# B&R Automation Studio project NAEUL004C00R13L518F00 (part 72)

#### Act_InitLocal.st
```iecst
(** 2019-04-16 **)
ACTION Act_InitLocal:

	//Input Reference Link To Local Variable
	p_udiRstErr ACCESS ADR(udiRstErr);
	p_bEn ACCESS ADR(bEn);
	p_bDis ACCESS ADR(bDis);
	p_bRun ACCESS ADR(bRun);
	p_bStop ACCESS ADR(bStop);
	p_bStep ACCESS ADR(bStep);

	p_sProgNm ACCESS ADR(sProgNm);
	p_bNtSettingsLoadDone ACCESS ADR(bNtSettingsLoadDone);

	p_usiMagConv ACCESS ADR(usiMagConv);
	p_bInfoEn ACCESS ADR(bInfoEn);

	pa_bMagDis ACCESS ADR(a_bMagDis);
	pa_bMagRej ACCESS ADR(a_bMagRej);
	p_bUSAllow ACCESS ADR(bUSAllow);

	p_bAllwChgWidth  ACCESS ADR(bAllwChgWidth);
	p_bAllwChgSlot ACCESS ADR(bAllwChgSlot);

	p_bNewMag ACCESS ADR(bNewMag);
	p_bRlsMag ACCESS ADR(bRlsMag);

	p_bConvInitDone ACCESS ADR(bConvInitDone);
	p_bConvHvBrd ACCESS ADR(bConvHvBrd);
	p_bConvGdBrd ACCESS ADR(bConvGdBrd);

	p_tyBufferStat1 ACCESS ADR(tyBufferStat1);
	p_tyBufferStat2 ACCESS ADR(tyBufferStat2);
	p_tyBufferStat3 ACCESS ADR(tyBufferStat3);

	p_bMagClampRS1 ACCESS ADR(bMagClampRS1);
	p_bMagClampRS2 ACCESS ADR(bMagClampRS2);
	p_bMagClampRS3 ACCESS ADR(bMagClampRS3);

	p_bMagEntrySen1 ACCESS ADR(bMagEntrySen1);
	p_bMagEntrySen2 ACCESS ADR(bMagEntrySen2);
	p_bMagEntrySen3 ACCESS ADR(bMagEntrySen3);

	p_bMagPresentSen1 ACCESS ADR(bMagPresentSen1);
	p_bMagPresentSen2 ACCESS ADR(bMagPresentSen2);
	p_bMagPresentSen3 ACCESS ADR(bMagPresentSen3);

	p_bBufferMagPresent1 ACCESS ADR(bBufferMagPresent1);
	p_bBufferMagPresent2 ACCESS ADR(bBufferMagPresent2);
	p_bBufferMagPresent3 ACCESS ADR(bBufferMagPresent3);

	p_dtBufferMagPresentTm1 ACCESS ADR(dtBufferMagPresentTm1);
	p_dtBufferMagPresentTm2 ACCESS ADR(dtBufferMagPresentTm2);
	p_dtBufferMagPresentTm3 ACCESS ADR(dtBufferMagPresentTm3);

	p_eBufferStat ACCESS ADR(eBufferStat);
	p_eBufferStatus ACCESS ADR(eBufferStatus);

	p_eMagConv2ClpStat ACCESS ADR(eMagConv2ClpStat);
	p_eMagConv2ClpStatus ACCESS ADR(eMagConv2ClpStatus);
	p_bMagConv2ClpHvMag ACCESS ADR(bMagConv2ClpHvMag);

	p_eUSSMEMAStat ACCESS ADR(eUSSMEMAStat);
	p_eUSSMEMAStatus ACCESS ADR(eUSSMEMAStatus);
	p_bUSSMEMATransporting ACCESS ADR(bUSSMEMATransporting);
	p_bUSSMEMAConvStart ACCESS ADR(bUSSMEMAConvStart);
	p_bUSSMEMAConvStop ACCESS ADR(bUSSMEMAConvStop);

	p_eAGVMagStat ACCESS ADR(eAGVMagStat);
	p_eAGVMagStatus ACCESS ADR(eAGVMagStatus);
	p_bAGVMagMcRunRdy ACCESS ADR(bAGVMagMcRunRdy);
	p_tyAGVToDTMag ACCESS ADR(tyAGVToDualMag);

	p_dtOpsMagConvUL3AcptTm ACCESS ADR(dtMagConvAcptTm);
	p_iOpsMagConvUL3MESAcptCond ACCESS ADR(iMagMESAcptCond);
END_ACTION
```

#### Act_Link.st
```iecst
(** 2018-12-11 **)
ACTION Act_Link:

	//Clamp RS
	p_bMagClampRS1 		:= (p_bLinkFixedMagClampRS1 AND p_bLinkRmtMagClampRS1) OR p_bLinkNewMagVerified1;
	p_bMagClampRS2		:= (p_bLinkFixedMagClampRS2 AND p_bLinkRmtMagClampRS2) OR p_bLinkNewMagVerified2;
	p_bMagClampRS3		:= (p_bLinkFixedMagClampRS3 AND p_bLinkRmtMagClampRS3) OR bNewMagVerified;

	//Mag Exchange Mode
	CASE p_eLinkMcParamMagExMode OF
		McSetMagXcAutoManMode:
			bMagManEx := TRUE;
			bMagAutoEx := TRUE;

		McSetMagXcAutoMode:
			bMagManEx := FALSE;
			bMagAutoEx := TRUE;

		McSetMagXcManMode:
			bMagManEx := TRUE;
			bMagAutoEx := FALSE;

	END_CASE

	//New magazine auto detection at inlet sensor
	fbMagAutoDetTm(IN := p_bLinkDIMagEntrySen OR p_bLinkDIMagPresentSen3, PT := DINT_TO_TIME(p_bLinkMcParamMagAutoDetTm));
	IF fbMagAutoDetTm.Q AND bMagManEx THEN
		bNewMagAutoDetected := TRUE;
	ELSE
		bNewMagAutoDetected := FALSE;
	END_IF

	IF p_bLinkNtParamMagModelAutoVerify THEN
		IF p_bLinkMagRcpCurrRcpMagModel = 0  //CAB706.2
			AND p_bDIMagConvHeightSen = TRUE
			AND p_bDIMagConvSelUnclampRS = FALSE
			AND p_bDIMagConvCAB717Sen = FALSE
			AND p_bDIMagConvSmallSen
			AND ((NOT p_bMagAWCloseLimit AND NOT  p_bMagAWOpenLimit) OR p_tyBufferStat3.bBffrMty = FALSE)
			THEN
			bNewMagVerified:= TRUE;

		ELSIF  p_bLinkMagRcpCurrRcpMagModel = 1 //CAB716.2
			AND p_bDIMagConvHeightSen = FALSE
			AND p_bDIMagConvSelUnclampRS = FALSE
			AND p_bDIMagConvCAB717Sen = FALSE
			AND p_bDIMagConvSmallSen
			AND ((NOT p_bMagAWCloseLimit AND NOT  p_bMagAWOpenLimit) OR p_tyBufferStat3.bBffrMty = FALSE)
			THEN
			bNewMagVerified:= TRUE;

		ELSIF  p_bLinkMagRcpCurrRcpMagModel = 2 //CAB717.2
			AND p_bDIMagConvHeightSen = FALSE
			AND p_bDIMagConvSelUnclampRS
			AND p_bDIMagConvCAB717Sen
			AND p_bDIMagConvLargeSen
			AND ((NOT p_bMagAWCloseLimit AND NOT  p_bMagAWOpenLimit) OR p_tyBufferStat3.bBffrMty = FALSE)
			THEN
			bNewMagVerified:= TRUE;
		ELSE
			bNewMagVerified:= FALSE;
		END_IF
	ELSE
		bNewMagVerified:= TRUE;
	END_IF

	bAIVInPos := p_tyAGVToDTMag.bVEHInPos3 OR p_bDISOTRcv;

	IF p_bBufferMagRemoved THEN
		bManualUnloadMag := FALSE;
	END_IF

	IF bAutoRcpEn THEN
		p_bUSAllow :=  ( NOT(p_bNtParamAutoRcpF1ArbitraryType) AND NOT(p_bMagPropDiffBlk) ) AND
						(p_bNtParamAutoRcpF1ArbitraryType AND p_sProdRcpCurrRcp1Name = p_sProdRcpCurrRcp2Name)	;
		p_bAllwChgWidth := p_bChgMagWidth AND NOT(p_bNtParamAutoRcpF1ArbitraryType);
		p_bAllwChgSlot	:= p_bChgMagSlot AND NOT(p_bNtParamAutoRcpF1ArbitraryType);

	ELSE
		p_bUSAllow := p_sProdRcpCurrRcp1Name = p_sProdRcpCurrRcp2Name;
	END_IF

END_ACTION
```

#### Cyclic.st
```iecst
(** 2019-03-22 **)
PROGRAM _CYCLIC

	IF bInitDone = FALSE THEN
		bInitDone	:= TRUE;

		Act_InitLocal;
		Act_InitGlobal;

	ELSIF bInitialDone = FALSE THEN
		IF p_bNtSettingsLoadDone = TRUE THEN
			bInitialDone	:= TRUE;

			Act_Initial;
		END_IF

	ELSE

		Act_RstErr;
		Act_LinkEn;
		Act_Link;
		Act_Background;
		Act_Alarm;
		Act_AlarmInfo1;

	END_IF

END_PROGRAM
```

#### Init.st
```iecst
(** 2019-03-25 **)
PROGRAM _INIT

	(* Always Change If Project Change *)

	//Physical Configuration
	usiMagConv	:= 3;

	//Pass Address To Global Address For External Use
	//Action, State & Status

	//Alarm
	p_OpsMagConvUL3AlmData	:= ADR(tyAlmData);
	p_OpsMagConvUL3AlmData1	:= ADR(tyAlmData1);

	//Output
	p_OpsMagConvUL3StepTxt			:= ADR(sStepTxt);
	p_OpsMagConvUL3Paused			:= ADR(bPaused);

	p_OpsMagConvUL3BufferAct		:= ADR(eBufferAct);
	p_OpsMagConvUL3MagConv2ClpAct	:= ADR(eMagConv2ClpAct);
	p_OpsMagConvUL3USSMEMAAct		:= ADR(eUSSMEMAAct);
	p_OpsMagConvUL3AGVMagAct		:= ADR(eAGVMagAct);

	p_OpsMagConvUL3InitDone				:= ADR(bOpsInitDone);
	p_OpsMagConvUL3MagBffrAvl			:= ADR(bMagBffrAvl);
	p_OpsMagConvUL3NewMagAllw			:= ADR(bNewMagAllw);
	p_OpsMagConvUL3RlsMagAllw			:= ADR(bRlsMagAllw);
	p_OpsMagConvUL3EjectMESStep			:= ADR(bEjectMESStep); //MES
	p_OpsMagConvUL3EjectMagNotAllw		:= ADR(bEjectMagNotAllw); //MES
	p_OpsMagConvUL3StepMagExitedWait	:= ADR(bStepMagExitedWait);
	p_OpsMagConvUL3StepUSCom			:= ADR(bStepMagUSCom);
	p_OpsMagConvUL3StepPLCGrab			:= ADR(bStepPLCGrab);

	p_OpsMagConvUL3StepSelClampCtrl		:= ADR(eSelClampCtrl);
	p_OpsMagConvUL3NewMagVerified		:= ADR(bNewMagVerified);
	p_OpsMagConvUL3MagFullExit			:= ADR(bStepMagFullExit);
	p_OpsMagConvUL3IncorrectMagModel    := ADR(bIncorrectMagazineModel);
	p_OpsMagConvUL3MagSizeL    			:= ADR(bMagSizeLarge);

	p_OpsMagConvUL3SafetyBarAct			:= ADR(eSafetyBarAct);
	p_OpsMagConvUL3MagAWEngageAct		:= ADR(eMagAWEngageAct);
	p_OpsMagConvUL3MagAWAct				:= ADR(eMagAWAct);

	p_OpsMagConvUL3USSOTAct				:= ADR(eUSSOTAct);
	p_OpsMagConvUL3DSSOTAct				:= ADR(eDSSOTAct);

	p_OpsAGVCommRdy3					:= ADR(bAGVComm3Rdy);

	p_OpsMagConvUL3UnclmpDone			:= ADR(bPneuUnclmpDone);
	p_OpsMagConvUL3MagAllwGo			:= ADR(udiMagAllwGo);

	p_OpsMagConvUL3ReadRFID				:= ADR(bReadRFID);
	p_OpsMagConvUL3WriteRFID			:= ADR(bWriteRFID);
	p_OpsMagConvUL3AWDone			 	:= ADR(bStepOpsMagAWDone);
	p_OpsMagConvUL3SlotUpdtDone			:= ADR(bStepOpsPitchUpdated);
	(* Always Change If Project Change *)

	p_OpsMagConvUL3AcptTm				:= ADR(dtMagConvAcptTm);
	p_OpsMagConvUL3MESAcptCond 			:= ADR(iMagMESAcptCond);
	p_OpsMagConvUL3MagExitedWait 		:= ADR(bMagExitedWait);
END_PROGRAM
```

#### Act_OpsInitial.st - Do Not Change!!!
```iecst
(** 2019-01-16 **)
ACTION Act_OpsInitial:

	eOpsStep			:= MagConvULStepNA;
	eGotoOpsStep		:= MagConvULStepInitMag;

	bOpsInitDone		:= FALSE;
	bMagBffrAvl			:= FALSE;
	bNewMagAllw			:= FALSE;
	bRlsMagAllw			:= FALSE;
	bStepMagExitedWait	:= FALSE;
	bAGVComm3Rdy		:= FALSE;

END_ACTION
```

#### Act_OpsRun.st
```iecst
(** 2019-04-16 **)
ACTION Act_OpsRun:
	IF p_bOpsTravLifErrCmdUnclmp THEN //from travLif width chk error
		eMagConv2ClpAct :=	MagConv2ClpActStopClpr;

		IF (p_eMagConv2ClpStatus = Done AND p_eMagConv2ClpStat = MagConv2ClpActStopClpr) THEN

			eMagConv2ClpAct	:= MagConv2ClpActIdle;
			bPneuUnclmpDone := TRUE; //To TravLifUL
		END_IF
	END_IF

	Act_LogStep;

	IF eGotoOpsStep <> eOpsStep THEN

		fbWrongMagTm(IN:= FALSE);
		fbReadRFIDTO(IN:= FALSE);
		fbWriteRFIDTO(IN:= FALSE);
		CASE eGotoOpsStep OF
			MagConvULStepBffrStatChk:  //For Siemen, Enter Condition
				IF ((p_eCustomerReq = Siemens OR p_eCustomerReq = We_Fabricate) AND p_bMcParamMESEn) AND eOpsStep = MagConvULStepVerifyMag THEN
					IF ePrevStepBeforeMESStdBy = MagConvULStepMagExitMnl OR ePrevStepBeforeMESStdBy = MagConvULStepMagExitClampCtrl THEN
						eGotoOpsStep		:= MagConvULStepMagExtMESStdByChk;
						eOpsStep			:= MagConvULStepMagExtMESStdByChk;
					ELSIF  iMagMESAcptCond > 0 THEN
						eGotoOpsStep		:= MagConvULStepBffrStatChk;
						eOpsStep			:= MagConvULStepBffrStatChk;
					ELSIF iMagMESAcptCond < 0 THEN
						eGotoOpsStep		:= MagConvULStepMagExitClampCtrl;
						eOpsStep			:= MagConvULStepMagExitClampCtrl;
					ELSIF iMagMESAcptCond = 0 THEN
						eGotoOpsStep		:= MagConvULStepMagEntMESStdByChk;
						eOpsStep			:= MagConvULStepMagEntMESStdByChk;
					END_IF
				ELSE
					eOpsStep	:= eGotoOpsStep;
				END_IF
			MagConvULStepMagExitClampCtrl: //For Siemen, Bffr Full,Changover Mag, AGV Rdy,Reject Mag
				IF (p_eCustomerReq = Siemens AND p_bMcParamMESEn) AND (eOpsStep <> MagConvULStepMagExtMESStdByChk )
					AND (p_tyLocalBufferStat.bBffrFull OR pa_bMagChangeOverBlk[p_usiMagConv] = TRUE OR p_bDISOTAGVReady)
					AND NOT(iMagMESAcptCond < 0)THEN
					eOpsStep := MagConvULStepMagExtMESStdByChk;
					eGotoOpsStep := MagConvULStepMagExtMESStdByChk;
					ePrevStepBeforeMESStdBy := MagConvULStepMagExitClampCtrl;
				ELSE
					eOpsStep	:= eGotoOpsStep;
					ePrevStepBeforeMESStdBy	:= MagConvULStepNA;
				END_IF
			MagConvULStepMagExitMnl: //For Siemens, Manual Rls
				IF (p_eCustomerReq = Siemens AND p_bMcParamMESEn)
					AND (eOpsStep <> MagConvULStepMagExtMESStdByChk AND eOpsStep <> MagConvULStepMagFullDSComm
					AND eOpsStep <> MagConvULStepMagEntMESStdByChk AND eOpsStep <> MagConvULStepVerifyMag)
					THEN
					eOpsStep := MagConvULStepMagExtMESStdByChk;
					eGotoOpsStep := MagConvULStepMagExtMESStdByChk;
					ePrevStepBeforeMESStdBy := MagConvULStepMagExitMnl;
				ELSE
//					sStepTxt	:= 'Waiting for Shutter Close';
//					IF (p_bNtParamProjOutletShut3Prep AND p_bDIOutShutterClosedRS3) OR (NOT(p_bNtParamProjOutletShut3Prep) AND p_bDIOutShutterClosedRS) THEN
						eOpsStep	:= eGotoOpsStep;
						ePrevStepBeforeMESStdBy	:= MagConvULStepNA;
//					END_IF
				END_IF
			MagConvULStepSelClampCtrl:
				IF p_bMagOrientChkSenPrep THEN
					IF p_bMagHeightDetEn AND p_bMagHeightDetPrep THEN

						IF p_bMag3OrientationChkSen1 AND p_bMagHeightDetSen3 THEN // Magazine Type Check with height Detection Sensor
							eOpsStep := eGotoOpsStep;
						ELSE
							eMagConv2ClpAct :=	MagConv2ClpActStopClpr; //Unclamp First

							IF (p_eMagConv2ClpStatus = Done AND p_eMagConv2ClpStat = MagConv2ClpActStopClpr) THEN

								eMagConv2ClpAct	:= MagConv2ClpActIdle;

								eStatus		:= Error;
								udiStatus	:= 10011;	//Wrong Magazine Orientation Placed.
							END_IF
						END_IF

					ELSE

						IF p_bMag3OrientationChkSen1 AND NOT p_bMagHeightDetSen3 THEN //Without Check Height Detection Sensor
							eOpsStep := eGotoOpsStep;
						ELSE
							eMagConv2ClpAct :=	MagConv2ClpActStopClpr; //Unclamp First

							IF (p_eMagConv2ClpStatus = Done AND p_eMagConv2ClpStat = MagConv2ClpActStopClpr) THEN

								eMagConv2ClpAct	:= MagConv2ClpActIdle;

								eStatus		:= Error;
								udiStatus	:= 10011;	//Wrong Magazine Orientation Placed.
							END_IF
						END_IF

					END_IF
				ELSE
					eOpsStep	:= eGotoOpsStep;
				END_IF
			ELSE
				eOpsStep	:= eGotoOpsStep;

		END_CASE

	END_IF

	IF eOpsStep = eGotoOpsStep THEN

		IF bPaused = FALSE THEN

			CASE eOpsStep OF

				MagConvULStepInitMag:
					sStepTxt	:= 'Initializing Magazine';
					p_usiMagConv := 3;
					CASE p_usiMagConv OF
						1:
							p_tyLocalBufferStat ACCESS ADR(p_tyBufferStat1);
							p_bLocalMagEntrySen ACCESS ADR(p_bMagEntrySen1);
							p_bLocalBufferMagPresent ACCESS ADR(p_bBufferMagPresent1);
							p_dtLocalBufferMagPresentTm ACCESS ADR(p_dtBufferMagPresentTm1);
						2:
							p_tyLocalBufferStat ACCESS ADR(p_tyBufferStat2);
							p_bLocalMagEntrySen ACCESS ADR(p_bMagEntrySen2);
							p_bLocalBufferMagPresent ACCESS ADR(p_bBufferMagPresent2);
							p_dtLocalBufferMagPresentTm ACCESS ADR(p_dtBufferMagPresentTm2);
						3:
							p_tyLocalBufferStat ACCESS ADR(p_tyBufferStat3);
							p_bLocalMagEntrySen ACCESS ADR(p_bMagEntrySen3);
							p_bLocalBufferMagPresent ACCESS ADR(p_bBufferMagPresent3);
							p_dtLocalBufferMagPresentTm ACCESS ADR(p_dtBufferMagPresentTm3);
					END_CASE

//					IF bMagExitedWait THEN
//						eGotoOpsStep	:= MagConvULStepMagExitedWait;
//					ELSE
//						eGotoOpsStep	:= MagConvULStepInitMagConv;
//					END_IF

					IF p_bProjLifTravMnlLoad = FALSE THEN
						eGotoOpsStep	:= MagConvULStepInitAWPneu;
					ELSE
						eGotoOpsStep	:= MagConvULStepMagUSComm; //no roller
					END_IF
					bPaused	:= p_bStop OR p_bStep;

				MagConvULStepInitAWPneu:
					sStepTxt	:= 'Initializing Pneumatic';

					eSafetyBarAct	:= PneuActExt;
					eMagAWEngageAct	:= PneuActRet;

					IF (p_eSafetyBarStatus = Done AND p_eSafetyBarStat = PneuActExt) AND (p_eMagAWEngageStatus = Done AND p_eMagAWEngageStat = PneuActRet) THEN
						eSafetyBarAct	:= PneuActIdle;
						eMagAWEngageAct	:= PneuActIdle;
						IF bMagExitedWait AND  ePrevExitStep = MagConvULStepMagExitMnl THEN
							//	eDSSOTAct	:= SOTActRun;
							eGotoOpsStep		:= MagConvULStepMagExitedWait; //sucessful exited
						ELSIF ePrevExitStep = MagConvULStepMagExitMnl  THEN
							eGotoOpsStep	:= MagConvULStepInitMagEnt; //halfway exiting, if magazine gone, init step
//						ELSIF  THEN
//							eGotoOpsStep	:= MagConvULStepMagExitClampCtrl; //want to exit before clamping
						ELSE
							eGotoOpsStep	:= MagConvULStepInitMagConv;
						END_IF
					END_IF

				MagConvULStepInitMagEnt:
					sStepTxt	:= 'Initializing Magazine Conveyor';
					eMagConv2ClpAct	:= MagConv2ClpActInit;
					IF (p_eMagConv2ClpStatus = Done AND p_eMagConv2ClpStat = MagConv2ClpActInit) THEN
						eMagConv2ClpAct	:= MagConv2ClpActIdle;
						IF p_bMagConv2ClpHvMag = FALSE THEN
							eGotoOpsStep	:= MagConvULStepMagUSComm;
							ePrevExitStep 		:= MagConvULStepNA;
							iMagMESAcptCond 	:= 0;
						ELSE
							eGotoOpsStep	:= MagConvULStepInitMagFixClp;
						END_IF
					END_IF

				MagConvULStepInitMagFixClp:
					sStepTxt	:= 'Initializing Fixed Clamp';
					eMagConv2ClpAct	:= MagConv2ClpActFixClprClamp;
					IF (p_eMagConv2ClpStatus = Done AND p_eMagConv2ClpStat = MagConv2ClpActFixClprClamp) THEN
							eMagConv2ClpAct	:= MagConv2ClpActIdle;
						IF bMagAutoEx THEN
							eDSSOTAct	:= SOTActRun;
						ELSE
							eDSSOTAct	:= SOTActIdle;
						END_IF

						IF p_bDIMagConvCAB717Sen THEN
							bMagSizeLarge := TRUE;
						ELSE
							bMagSizeLarge := FALSE;
						END_IF
							eGotoOpsStep	:= MagConvULStepSelClampCtrl;
					END_IF

				MagConvULStepInitMagConv:
					sStepTxt	:= 'Initializing Magazine Conveyor';

					eMagConv2ClpAct	:= MagConv2ClpActInitStopClp;
					eSelClampCtrl := PneuActExt;

					IF (p_eMagConv2ClpStatus = Done AND p_eMagConv2ClpStat = MagConv2ClpActInitStopClp)
						AND (p_eSelClampCtrlStat = PneuActExt AND p_eSelClampCtrlStatus = Done)
						THEN
						eSelClampCtrl := PneuActIdle;
						eMagConv2ClpAct	:= MagConv2ClpActIdle;

						IF p_bMagConv2ClpHvMag = FALSE THEN
							eGotoOpsStep	:= MagConvULStepMagUSComm;
							ePrevExitStep 		:= MagConvULStepNA;
							iMagMESAcptCond 	:= 0;
						ELSE
							//	eGotoOpsStep	:= MagConvULStepBffrStatChk;
							eGotoOpsStep	:= MagConvULStepSelClampCtrl;
						END_IF

						bPaused	:= p_bStop OR p_bStep;
					END_IF

				MagConvULStepMagUSComm:
					sStepTxt	:= 'Communicating AIV And Ready For Transport In Magazine';

					eAGVMagAct	:= AGVMagActEnter;
					IF bMagAutoEx THEN
						eUSSOTAct	:= SOTActRun;
					ELSE
						eUSSOTAct	:= SOTActIdle;
					END_IF

					eDSSOTAct	:= SOTActIdle;
					bMagSizeLarge := FALSE;
					bMagExitedWait	:= FALSE;

					IF p_bSafetyBarExtended = FALSE THEN
						eGotoOpsStep	:= MagConvULStepSafetyBarExt;
					ELSIF p_bAGVMagMcRunRdy = TRUE OR p_bUSSOTTransporting= TRUE THEN
						eGotoOpsStep	:= MagConvULStepMagEnt;

					ELSIF p_bNewMag = TRUE OR bNewMagAutoDetected = TRUE THEN
						eAGVMagAct		:= AGVMagActIdle;
						eGotoOpsStep	:= MagConvULStepMagEntMnl;

					ELSE
						bPaused	:= p_bStop;

						IF bPaused = TRUE THEN
							eAGVMagAct	:= AGVMagActIdle;
							eUSSOTAct	:= SOTActIdle;
						END_IF

					END_IF

				MagConvULStepMagEnt:

					IF p_bUSSOTConvStart THEN
						sStepTxt	:= 'Conveyor Entering Magazine To End';
						eMagConv2ClpAct	:= MagConv2ClpActEntStopClp;

					ELSIF bNewMagAutoDetected = TRUE THEN
						eAGVMagAct			:= AGVMagActIdle;
						eGotoOpsStep		:= MagConvULStepMagEntMnl;

					ELSIF p_bUSSOTConvStop THEN
						sStepTxt	:= 'Conveyor Stopping';
						eMagConv2ClpAct	:= MagConv2ClpActStopClpr;
						IF (p_eMagConv2ClpStatus = Done AND p_eMagConv2ClpStat = MagConv2ClpActStopClpr) THEN
							eMagConv2ClpAct		:= MagConv2ClpActIdle;

						END_IF
					END_IF

					IF (p_eMagConv2ClpStatus = Done AND p_eMagConv2ClpStat = MagConv2ClpActEntStopClp) THEN
						eAGVMagAct			:= AGVMagActIdle;
						eMagConv2ClpAct		:= MagConv2ClpActIdle;
						eUSSOTAct			:= SOTActIdle;
						eGotoOpsStep		:= MagConvULStepSelClampCtrl;
						bPaused	:= p_bStop OR p_bStep;

					ELSE

					END_IF

				MagConvULStepMagEntMnl:
					sStepTxt	:= 'Magazine Conveyor Entering Magazine Manually';

					IF p_bProjLifTravMnlLoad = FALSE THEN
						eMagConv2ClpAct	:= MagConv2ClpActEntStopClp;
					ELSE
						eGotoOpsStep	:= MagConvULStepSelClampCtrl; //no roller
					END_IF

					IF p_eMagConv2ClpStatus = Done AND p_eMagConv2ClpStat = MagConv2ClpActEntStopClp THEN
						eMagConv2ClpAct	:= MagConv2ClpActIdle;
						//	eGotoOpsStep	:= MagConvULStepBffrStatChk;
							eGotoOpsStep	:= MagConvULStepSelClampCtrl;
						eUSSOTAct			:= SOTActIdle;
						eAGVMagAct			:= AGVMagActIdle;
						bPaused	:= p_bStop OR p_bStep;
					END_IF

				MagConvULStepSelClampCtrl:
					sStepTxt	:= 'Magazine Selection Control';
					bNewMagVerifyStarted := TRUE;

					CASE p_bLinkMagRcpCurrRcpMagModel OF
						0: //CAB706.2
							IF p_bDIMagConvCAB717Sen = FALSE THEN
								eSelClampCtrl := PneuActRet;
							END_IF

							eGotoOpsStep		:= MagConvULStepVerifyMag;

						1: //CAB716.2
							IF p_bDIMagConvCAB717Sen = FALSE THEN
								eSelClampCtrl := PneuActRet;
							END_IF

							eGotoOpsStep		:= MagConvULStepVerifyMag;

						2: //CAB717.2
							eSelClampCtrl := PneuActExt;

							eGotoOpsStep	:= MagConvULStepVerifyMag;

					END_CASE

					bPaused	:= p_bStop OR p_bStep;

				MagConvULStepVerifyMag:
					sStepTxt	:= 'Magazine Model Verification';

					bNewMagVerifyStarted := TRUE;
					fbWrongMagTm(IN:= bNewMagVerified = FALSE);
					IF fbWrongMagTm.Q AND NOT bMagExitedWait THEN
						fbWrongMagTm(IN:= FALSE);
						eGotoOpsStep		:= MagConvULStepMagExitMnl;
					ELSIF ePrevExitStep = MagConvULStepMagExitMnl THEN
						eGotoOpsStep		:= MagConvULStepMagExitMnl;
					ELSIF ePrevExitStep = MagConvULStepMagExitClampCtrl THEN
						eGotoOpsStep		:= MagConvULStepMagExitClampCtrl;
					ELSIF bNewMagVerified  THEN
						eSelClampCtrl	:= PneuActIdle;

						eGotoOpsStep		:= MagConvULStepBffrStatChk; //to RFID scanning if applicable

					END_IF

					IF p_bDIMagConvCAB717Sen THEN
						bMagSizeLarge := TRUE;
					ELSE
						bMagSizeLarge := FALSE;
					END_IF

					IF p_bSelfTest THEN
						eGotoOpsStep	:= MagConvULStepMagCmp;
					END_IF

					bPaused	:= p_bStop OR p_bStep;

				MagConvULStepMagEntMESStdByChk:
					IF p_eCustomerReq = Siemens THEN
						sStepTxt	:= 'Read RFID Chk step';
					ELSE
						sStepTxt	:= 'Wait for MES feedback';
					END_IF
					bReadRFID := TRUE;
					fbReadRFIDTO(IN:= bReadRFID,PT := DINT_TO_TIME(p_diMcParamMESResponseTO));
					iMagMESAcptCond := (p_tyResponseFromMES.iAcceptCondition);
					IF p_tyResponseFromMES.iAcceptCondition > 0  THEN //Accept
						eGotoOpsStep := MagConvULStepBffrStatChk;
						dtMagConvAcptTm	:= p_dtCurrDT;
					ELSIF p_tyResponseFromMES.iAcceptCondition < 0  THEN//No Accept
						eGotoOpsStep	:= MagConvULStepMagExitClampCtrl;
					ELSIF fbReadRFIDTO.Q AND p_bRlsMag THEN
						sStepTxt	:= 'Wait for Read RFID';;
						eGotoOpsStep := MagConvULStepMagExitMnl;
					END_IF
					IF eGotoOpsStep <> MagConvULStepMagEntMESStdByChk THEN
						bReadRFID := FALSE;
						fbReadRFIDTO(IN:= bReadRFID);

					END_IF
					bPaused	:= p_bStop OR p_bStep;

				MagConvULStepBffrStatChk:
					sStepTxt	:= 'Checking Buffer Status';

					IF p_eBufferStatus = Idle THEN

						IF p_tyLocalBufferStat.bBffrFull = TRUE
							//AND p_bOutShutterExtended
							THEN
							//	eGotoOpsStep	:= MagConvULStepMagFullDSComm;
							eGotoOpsStep	:= MagConvULStepMagExitClampCtrl;
						ELSE
		//	20210420		eGotoOpsStep	:= MagConvULStepMagCmp;
							eGotoOpsStep	:= MagConvULStepSafetyBarRet;
						END_IF

						bPaused	:= p_bStop OR p_bStep;

					END_IF

				MagConvULStepChkMag:

					sStepTxt	:= 'Checking Magazine Status';
//					IF p_bSafetyBarExtended = FALSE THEN
//							eGotoOpsStep	:= MagConvULStepSafetyBarExt;

//					ELSIF p_bMagPresentSen1 = TRUE THEN
					IF p_bMagPresentSen = TRUE THEN
						IF p_tyLocalBufferStat.bBffrMty = TRUE THEN
							//Buffer Empty
							IF  bAutoRcpEn THEN //NOT(p_bUSAllow) AND
								eGotoOpsStep	:= MagConvULStepMagCmp;
							ELSIF bMagAWDone = FALSE THEN
								eGotoOpsStep	:= MagConvULStepMagAWEngage;
//							ELSIF p_bSafetyBarRetracted = FALSE THEN
//								eGotoOpsStep	:= MagConvULStepSafetyBarRet;
							ELSE
								eGotoOpsStep	:= MagConvULStepMagCmp;
							END_IF

						ELSIF p_tyLocalBufferStat.bBffrFull = TRUE
						//	AND p_bOutShutterExtended
							THEN
							//Buffer Full

							IF p_bSafetyBarExtended = FALSE THEN
								eGotoOpsStep	:= MagConvULStepSafetyBarExt;
							ELSE
								eGotoOpsStep    := MagConvULStepMagExitClampCtrl;
							END_IF

						ELSE
							//Buffer Available
//							IF p_bSafetyBarRetracted = FALSE THEN
//								eGotoOpsStep	:= MagConvULStepSafetyBarRet;
//							ELSE
								eGotoOpsStep	:= MagConvULStepMagCmp;
//							END_IF

						END_IF

					ELSE

//						IF p_bSafetyBarExtended = FALSE THEN
//							eGotoOpsStep	:= MagConvULStepSafetyBarExt;
//						ELSE
							eGotoOpsStep	:= MagConvULStepMagUSComm;
//						END_IF

					END_IF

					bPaused	:= p_bStop OR p_bStep;

				MagConvULStepSafetyBarExt:
					sStepTxt	:= 'Extending Safety Bar';

					eSafetyBarAct	:= PneuActExt;

					IF p_eSafetyBarStatus = Done AND p_eSafetyBarStat = PneuActExt THEN
						eSafetyBarAct	:= PneuActIdle;
						eGotoOpsStep	:= MagConvULStepChkMag;

						bPaused	:= p_bStop OR p_bStep;
					END_IF

				MagConvULStepSafetyBarRet:
					sStepTxt	:= 'Retracting Safety Bar';

					eSafetyBarAct	:= PneuActRet;

					IF p_eSafetyBarStatus = Done AND p_eSafetyBarStat = PneuActRet THEN
						eSafetyBarAct	:= PneuActIdle;
					//	eGotoOpsStep	:= MagSetupULStepMagNBffrStatChk;
						eGotoOpsStep	:= MagConvULStepChkMag;

						bPaused	:= p_bStop OR p_bStep;
					END_IF

				MagConvULStepMagAWEngage:
					sStepTxt	:= 'Engaging Magazine Auto Width';

					eMagAWAct	:= MagAWActEngage;

					IF p_bMagAWEngaging = TRUE THEN
						eMagAWEngageAct	:= PneuActExt;
					END_IF

					IF (p_eMagAWStatus = Done AND p_eMagAWStat = MagAWActEngage) AND (p_eMagAWEngageStatus = Done AND p_eMagAWEngageStat = PneuActExt) THEN
						eMagAWAct		:= MagAWActIdle;
						eMagAWEngageAct	:= PneuActIdle;
						eGotoOpsStep	:= MagConvULStepMagAWHm;
						bPaused	:= p_bStop OR p_bStep;

					END_IF

				MagConvULStepMagAWHm:
					sStepTxt	:= 'Homing Magazine Auto Width';

					eMagAWAct	:= MagAWActHoming;

					IF p_eMagAWStatus = Done AND p_eMagAWStat = MagAWActHoming THEN
						eMagAWAct		:= MagAWActIdle;
						eGotoOpsStep	:= MagConvULStepMagAWMov;

					ELSIF p_bMagAWErr THEN

						eStatus			:= Error;
						udiStatus		:= 10009;
					END_IF

				MagConvULStepMagAWMov:
					sStepTxt	:= 'Moving Magazine Auto Width';

					eMagAWAct	:= MagAWActGoWidthOff;

					IF p_eMagAWStatus = Done AND p_eMagAWStat = MagAWActGoWidthOff THEN
						bMagAWDone		:= TRUE;
						eMagAWAct		:= MagAWActIdle;
						eGotoOpsStep	:= MagConvULStepMagAWDisengage;

						bPaused	:= p_bStop OR p_bStep;

					ELSIF p_bMagAWErr THEN

						eStatus			:= Error;
						udiStatus		:= 10009;
					END_IF

				MagConvULStepMagAWDisengage:
					sStepTxt	:= 'Disengaging Magazine Auto Width';

					eMagAWEngageAct	:= PneuActRet;

					IF p_eMagAWEngageStatus = Done AND p_eMagAWEngageStat = PneuActRet THEN
						eMagAWEngageAct	:= PneuActIdle;

						eGotoOpsStep	:= MagConvULStepSafetyBarRet;

						bPaused	:= p_bStop OR p_bStep;
					END_IF

				MagConvULStepMagCmp:
					sStepTxt	:= 'Comparing Magazine';

					a_tyMagAllwBffrStat[1]	:= p_tyBufferStat1;
					a_tyMagAllwBffrStat[2]	:= p_tyBufferStat2;
					a_tyMagAllwBffrStat[3]	:= p_tyBufferStat3;

					a_bMagAllwMagClamped[1]	:= p_bMagClampRS1 ;
					a_bMagAllwMagClamped[2]	:= p_bMagClampRS2 ;
					a_bMagAllwMagClamped[3]	:= p_bMagClampRS3 ;

					a_bMagAllwMagPresent[1]	:= p_bBufferMagPresent1 AND NOT(p_bOpsMagConvUL1MagExitedWait);
					a_bMagAllwMagPresent[2]	:= p_bBufferMagPresent2 AND NOT(p_bOpsMagConvUL2MagExitedWait);
					a_bMagAllwMagPresent[3]	:= p_bBufferMagPresent3 AND NOT(bMagExitedWait);

					IF NOT(bAutoRcpEn AND p_bMcParamMESEn) THEN
						a_udiMagAllwMagPresentTm[1]	:= DT_TO_UDINT(p_dtBufferMagPresentTm1);
						a_udiMagAllwMagPresentTm[2]	:= DT_TO_UDINT(p_dtBufferMagPresentTm2);
						a_udiMagAllwMagPresentTm[3]	:= DT_TO_UDINT(p_dtBufferMagPresentTm3);
					ELSE
						a_udiMagAllwMagPresentTm[1]	:= DT_TO_UDINT(p_dtOpsMagConvUL1AcptTm);
						a_udiMagAllwMagPresentTm[2]	:= DT_TO_UDINT(p_dtOpsMagConvUL2AcptTm);
						a_udiMagAllwMagPresentTm[3]	:= DT_TO_UDINT(p_dtOpsMagConvUL3AcptTm);

						a_iMagMESAcptCond[1] := p_iOpsMagConvUL1MESAcptCond;
						a_iMagMESAcptCond[2] := p_iOpsMagConvUL2MESAcptCond;
						a_iMagMESAcptCond[3] := p_iOpsMagConvUL3MESAcptCond;
					END_IF

					//Sorting Priority
					memset(ADR(a_udiMagAllwPriority), 0, SIZEOF(a_udiMagAllwPriority));

					FOR udi := 1 TO 3 DO
						udiCount	:= 3;
						udiCmpTm	:= a_udiMagAllwMagPresentTm[udi];

						FOR udi1 := 1 TO 3 DO
							IF a_udiMagAllwMagPresentTm[udi1] < udiCmpTm THEN
								udiCount	:= udiCount - 1;
							END_IF
						END_FOR

						a_udiMagAllwPriority[udi]	:= udiCount;
					END_FOR

//					FOR udi := 3 TO 1 BY -1 DO
//						FOR udi1 := 3 TO 1 BY -1 DO
//							IF (udi <> udi1) AND (a_udiMagAllwPriority[udi] = a_udiMagAllwPriority[udi1]) THEN
//								a_udiMagAllwPriority[udi1]	:= a_udiMagAllwPriority[udi1] - 1;
//							END_IF
//						END_FOR
//					END_FOR

					//Checking Buffer Status
					memset(ADR(a_udiMagAllwSum), 0, SIZEOF(a_udiMagAllwSum));

					FOR udi := 1 TO 3 DO
						//Priority
						a_udiMagAllwSum[udi]	:= a_udiMagAllwSum[udi] + a_udiMagAllwPriority[udi];
						//Enable
						IF pa_bMagDis[udi] = FALSE THEN
							a_udiMagAllwSum[udi]	:= a_udiMagAllwSum[udi] + 1000;
						END_IF
						//Magazine Clamped
						IF a_bMagAllwMagClamped[udi] = TRUE THEN
							a_udiMagAllwSum[udi]	:= a_udiMagAllwSum[udi] + 1000;
						END_IF
						//Magazine Present
						IF a_bMagAllwMagPresent[udi] = TRUE THEN
							a_udiMagAllwSum[udi]	:= a_udiMagAllwSum[udi] + 1000;
						END_IF
						//Magazine Empty
						IF a_tyMagAllwBffrStat[udi].bBffrMty = TRUE THEN
							a_udiMagAllwSum[udi]	:= a_udiMagAllwSum[udi] + 2500;
						END_IF
						//Magazine Available
						IF a_tyMagAllwBffrStat[udi].bBffrFull = FALSE AND a_tyMagAllwBffrStat[udi].bBffrMty = FALSE THEN
							a_udiMagAllwSum[udi]	:= a_udiMagAllwSum[udi] + 3000;
						END_IF
						//Magazine Reject
						IF pa_bMagRej[udi] = TRUE THEN
							a_udiMagAllwSum[udi]	:= a_udiMagAllwSum[udi] + 6000;
						END_IF
						//Customized Width Change
						IF bAutoRcpEn THEN
							IF pa_bMagChangeOverBlk[udi] = TRUE  THEN
								a_udiMagAllwSum[udi]	:= a_udiMagAllwSum[udi] - 1000;
							END_IF
							IF  p_bMcParamMESEn THEN
								IF a_iMagMESAcptCond[udi] = 0 AND  a_bMagAllwMagPresent [udi] THEN
									a_udiMagAllwSum[udi]	:= a_udiMagAllwSum[udi] - 1000;
								END_IF
							END_IF
						END_IF
					END_FOR

					udiMagAllwGo	:= 99;

					FOR udi := 1 TO 3 DO
						IF (a_udiMagAllwSum[udi] >= 6000 AND a_udiMagAllwSum[udi] < 7000 AND pa_bMagRej[usiMagConv] = FALSE)	//Enable + Magazine Clamped + Magazine Present + Magazine Available
							OR (a_udiMagAllwSum[udi] >= 12000 AND pa_bMagRej[usiMagConv] = TRUE) THEN							//Reject + Enable + Magazine Clamped + Magazine Present + Magazine Available

							IF udiMagAllwGo <> 99 THEN
								//Priority
								IF a_udiMagAllwSum[udi] > a_udiMagAllwSum[udiMagAllwGo] THEN
									udiMagAllwGo	:= udi;
								END_IF
							ELSE
								udiMagAllwGo	:= udi;
							END_IF

						END_IF

					END_FOR

					IF udiMagAllwGo = 99 THEN

						FOR udi := 1 TO 3 DO
							IF (a_udiMagAllwSum[udi] >= 5500 AND a_udiMagAllwSum[udi] < 7000 AND pa_bMagRej[usiMagConv] = FALSE)	//Enable + Magazine Clamped + Magazine Present + Magazine Empty
								OR (a_udiMagAllwSum[udi] >= 11500 AND pa_bMagRej[usiMagConv] = TRUE) THEN							//Reject + Enable + Magazine Clamped + Magazine Present + Magazine Empty

								IF udiMagAllwGo <> 99 THEN
									//Priority
									IF a_udiMagAllwSum[udi] > a_udiMagAllwSum[udiMagAllwGo] THEN
										udiMagAllwGo	:= udi;
									END_IF
								ELSE
									udiMagAllwGo	:= udi;
								END_IF

							END_IF

						END_FOR

					END_IF

					IF p_bRlsMag = TRUE THEN
						eGotoOpsStep	:= MagConvULStepMagExitMnl;
					ELSIF (p_bDISOTAGVReady OR
						pa_bMagChangeOverBlk[p_usiMagConv] )
						AND (p_eCustomerReq = Siemens OR p_eCustomerReq = We_Fabricate )THEN
						eGotoOpsStep	:= MagConvULStepMagExitClampCtrl;
					ELSIF p_tyLocalBufferStat.bBffrFull = TRUE AND p_bOutShutterExtended OR (p_bUSAllow = FALSE AND NOT(bAutoRcpEn)) THEN //in normal mode, when change Rcp, mean Eject all magazine
					//	eGotoOpsStep    := MagConvULStepMagFullDSComm;
						eGotoOpsStep	:= MagConvULStepMagExitClampCtrl;
					ELSIF NOT(p_bUSAllow) AND bAutoRcpEn  AND  udiMagAllwGo = p_usiMagConv THEN
						//do nothing when blocking
						sStepTxt	:= 'Comparing Mag: Waiting available magazine to change width';
						bPaused	:= p_bStop;
					ELSIF p_bAllwChgWidth AND bAutoRcpEn THEN
						eGotoOpsStep	:= 	MagConvULStepMagAWEngage;
					ELSIF p_bAllwChgSlot AND bAutoRcpEn THEN
						eGotoOpsStep	:= 	MagConvULStepMtyBffr; //MagConvULStepMagAWEngage;

					ELSE

						IF (p_bUSAllow = TRUE) AND (udiMagAllwGo <> 99) THEN

							IF udiMagAllwGo = p_usiMagConv THEN
								bMagBffrAvl		:= TRUE;
//								IF NOT(bAutoRcpEn AND p_tyLocalBufferStat.bBffrMty = TRUE) THEN
									eGotoOpsStep	:= MagConvULStepNxtLoadBffr;
//								ELSE
//									eGotoOpsStep	:= MagConvULStepMtyBffr;
//								END_IF;

								bPaused	:= p_bStop OR p_bStep;
							ELSE
								bPaused	:= p_bStop;
							END_IF

						ELSE
							bPaused	:= p_bStop;
						END_IF

					END_IF
				MagConvULStepMtyBffr:
					sStepTxt	:= 'Resetting Buffer Setting';
					eBufferAct := BufferActSetMty;

					IF p_eBufferStatus = Done AND p_eBufferStat = BufferActSetMty THEN
						eBufferAct		:= BufferActIdle;
						eGotoOpsStep	:= MagConvULStepMagCmp;

						bPaused	:= p_bStop OR p_bStep;
					END_IF

				MagConvULStepNxtLoadBffr:
					sStepTxt	:= 'Computing Next Load Buffer';

					eBufferAct	:= BufferActNxtLoad;

					IF p_eBufferStatus = Done AND p_eBufferStat = BufferActNxtLoad THEN
						eBufferAct		:= BufferActIdle;
						eGotoOpsStep	:= MagConvULStepBffrUSComm;

						bPaused	:= p_bStop OR p_bStep;
					END_IF

				MagConvULStepBffrUSComm:
					sStepTxt	:= 'Communicating Buffer Upstream';

					eUSSMEMAAct	:= SMEMAActRun;

					IF p_bUSSMEMATransporting = TRUE THEN
						eGotoOpsStep	:= MagConvULStepBffrEntBrd;
						IF p_eNtParamProjMagBuffferActLoad = BufferActLoadWhenStarted
							THEN

							eBufferAct	:= BufferActLoad;
						END_IF
					ELSIF p_bRlsMag = TRUE AND (p_bOpsTravLifAllwExitMag OR p_eCustomerReq <> Siemens) THEN
						bMagBffrAvl		:= FALSE;
						eUSSMEMAAct		:= SMEMAActIdle;
						eGotoOpsStep	:= MagConvULStepMagExitMnl;

					ELSIF  ((p_bAllwChgWidth OR p_bAllwChgSlot) AND NOT(p_bMcParamAutoRcpDis) ) OR p_bUSAllow = FALSE THEN
						bMagBffrAvl		:= FALSE;
						eUSSMEMAAct		:= SMEMAActIdle;
						eGotoOpsStep	:= MagConvULStepMagCmp;

						bPaused	:= p_bStop OR p_bStep;

					ELSIF (p_tyLocalBufferStat.bBffrFull = TRUE ) //AND p_bOutShutterExtended OR p_eCustomerReq = Siemens
						OR (p_bDISOTAGVReady AND p_bOpsTravLifAllwExitMag) THEN //OR  p_bUSAllow = FALSE THEN
						bMagBffrAvl		:= FALSE;
						eUSSMEMAAct		:= SMEMAActIdle;
						//	eGotoOpsStep    := MagConvULStepMagFullDSComm;
						eGotoOpsStep    := MagConvULStepMagExitClampCtrl;
					ELSE

						IF pa_bMagDis[usiMagConv] = TRUE THEN		//Checking Magazine Enable
							bMagBffrAvl		:= FALSE;
							eGotoOpsStep	:= MagConvULStepMagCmp;

							bPaused	:= p_bStop OR p_bStep;
						ELSE
							bPaused	:= p_bStop;
						END_IF

						IF bPaused = TRUE OR pa_bMagDis[usiMagConv] = TRUE THEN
							eUSSMEMAAct	:= SMEMAActIdle;
						END_IF

					END_IF

				MagConvULStepBffrEntBrd:
					IF p_bUSSMEMATransporting AND EDGEPOS(p_bUSSMEMAConvStart) THEN
						sStepTxt	:= 'Transferring Board Into Magazine';
						IF p_eNtParamProjMagBuffferActLoad = BufferActLoadWhenStarted
							THEN

							eBufferAct	:= BufferActLoad;
						END_IF

					END_IF

					IF p_bUSSMEMATransporting AND EDGEPOS(p_bUSSMEMAConvStop) THEN
						sStepTxt	:= 'Stop Transferring';
						//Do Nothing
					END_IF

					//					IF p_bUSSMEMATransporting = FALSE
					//						THEN
					//						eGotoOpsStep	:= MagConvULStepBffrUSComm;
					//					END_IF

					IF (p_eUSSMEMAStatus = Done AND p_eUSSMEMAStat = SMEMAActRun)
						AND (p_eConvStat = ConvActExitPshr AND p_eConvStatus = Done)
						THEN
						eUSSMEMAAct		:= SMEMAActIdle;
						eGotoOpsStep	:= MagConvULStepLoadBffr;
					END_IF

				MagConvULStepLoadBffr:
					sStepTxt	:= 'Loading Buffer';

					eBufferAct	:= BufferActLoad;

					IF p_eBufferStatus = Done AND p_eBufferStat = BufferActLoad THEN
						eBufferAct		:= BufferActIdle;
						bMagBffrAvl		:= FALSE;
						eGotoOpsStep	:= MagConvULStepBffrStatChk;

						bPaused	:= p_bStop OR p_bStep;
					END_IF
				MagConvULStepMagExtMESStdByChk:
					sStepTxt	:= 'Mag StdBy for MES response Before Exiting';
					bWriteRFID := TRUE;
					fbWriteRFIDTO(IN:= bWriteRFID,PT := DINT_TO_TIME(p_diMcParamMESResponseTO) );
					IF p_tyResponseFromMES.bRFIDWriteComplete  THEN //Accept
						IF ePrevStepBeforeMESStdBy = MagConvULStepMagExitMnl THEN
							eGotoOpsStep := MagConvULStepMagExitMnl;
						ELSIF ePrevStepBeforeMESStdBy = MagConvULStepMagExitClampCtrl THEN
							eGotoOpsStep := MagConvULStepMagExitClampCtrl;
						END_IF
					ELSIF fbWriteRFIDTO.Q  AND p_bRlsMag THEN
						sStepTxt	:= 'MES response to Write RFID Timeout, Press Rls Mag to Manual Exit ';

						eGotoOpsStep := MagConvULStepMagExitMnl;

					END_IF

					bPaused	:= p_bStop OR p_bStep;

				MagConvULStepMagExitClampCtrl:
					sStepTxt	:= 'Extending Selection Clamp';

					eSelClampCtrl := PneuActExt;
					eMagAWEngageAct	:= PneuActRet;
					ePrevExitStep := MagConvULStepMagExitClampCtrl;
					IF (p_eSelClampCtrlStat = PneuActExt AND p_eSelClampCtrlStatus = Done)
						OR (p_eMagAWEngageStat = PneuActRet AND p_eMagAWEngageStatus = Done)
						THEN
						eMagAWEngageAct	:= PneuActIdle;
						eSelClampCtrl	:= PneuActIdle;
						eGotoOpsStep    := MagConvULStepMagExitSafeBarCtrl;
						bPaused	:= p_bStop OR p_bStep;
					END_IF

				MagConvULStepMagExitSafeBarCtrl:
					IF p_bSafetyBarExtended = FALSE THEN
						eSafetyBarAct	:= PneuActExt;

						IF p_eSafetyBarStatus = Done AND p_eSafetyBarStat = PneuActExt THEN
							eSafetyBarAct	:= PneuActIdle;
							eGotoOpsStep    := MagConvULStepMagFullDSComm;

							bPaused	:= p_bStop OR p_bStep;
						END_IF
					ELSE
						eGotoOpsStep    := MagConvULStepMagFullDSComm;
					END_IF

				MagConvULStepMagFullDSComm:
					sStepTxt	:= 'Communicating AGV Machine And Ready Exit';

					eAGVMagAct	:= AGVMagActExit;
					IF bMagAutoEx THEN
						eDSSOTAct	:= SOTActRun;
					ELSE
						eDSSOTAct	:= SOTActIdle;
					END_IF

					IF p_bAGVMagMcRunRdy = TRUE THEN
						eGotoOpsStep	:= MagConvULStepMagFullExit;

					ELSIF p_bRlsMag = TRUE
						OR (p_tyLocalBufferStat.bBffrFull AND p_bDIOutShutterClosedRS3 ) //AND p_bOutShutterExtended )
						OR (pa_bMagChangeOverBlk[p_usiMagConv] = TRUE AND bAutoRcpEn)
						OR (p_bUSAllow = FALSE AND NOT(bAutoRcpEn) )THEN
						eAGVMagAct		:= AGVMagActIdle;
						eGotoOpsStep	:= MagConvULStepMagExitMnl;

					ELSE
						bPaused	:= p_bStop;

						IF bPaused = TRUE THEN
							eAGVMagAct	:= AGVMagActIdle;
						END_IF

					END_IF

				MagConvULStepMagFullExit:
					sStepTxt	:= 'Magazine Conveyor Exiting Magazine';

					eMagConv2ClpAct	:= MagConv2ClpActExitClpr;
					eSelClampCtrl	:= PneuActExt;

					IF ((p_eAGVMagStatus = Done AND p_eAGVMagStat = AGVMagActExit)
						OR (p_eDSSOTStatus = Done AND p_eDSSOTStat = SOTActRun))
						AND (p_eMagConv2ClpStatus = Done AND p_eMagConv2ClpStat = MagConv2ClpActExitClpr)
						AND (p_eSelClampCtrlStatus = Done AND p_eSelClampCtrlStat = PneuActExt)
						THEN
						eDSSOTAct			:= SOTActIdle;
						eAGVMagAct			:= AGVMagActIdle;
						eMagConv2ClpAct		:= MagConv2ClpActIdle;
						eSelClampCtrl		:= PneuActIdle;
						eGotoOpsStep		:= MagConvULStepMagExitedAGVWait;
						bMagSizeLarge := FALSE;
						bPaused	:= p_bStop OR p_bStep;
					END_IF

				MagConvULStepMagExitedAGVWait:
					sStepTxt  := 'Magazine Exited and wait for AGV Leave';

					IF bAIVInPos = FALSE OR p_bBufferMagRemoved THEN
						ePrevExitStep 		:= MagConvULStepNA;
						iMagMESAcptCond 	:= 0;
						eGotoOpsStep        := MagConvULStepMagUSComm;
						eDSSOTAct			:= SOTActIdle;

					END_IF

					bPaused   := p_bStop OR p_bStep;

				MagConvULStepMagExitMnl:
					sStepTxt	:= 'Magazine Conveyor Exiting Magazine Manually';
					IF p_bProjLifTravMnlLoad = FALSE THEN
						eMagConv2ClpAct	:= MagConv2ClpActPreExitClpr;
						eSelClampCtrl	:= PneuActExt;
						eSafetyBarAct	:= PneuActExt;
					ELSE
						eGotoOpsStep		:= MagConvULStepMagExitedWait; //no roller
					END_IF
					ePrevExitStep := MagConvULStepMagExitMnl;
					IF ((p_eMagConv2ClpStatus = Done AND p_eMagConv2ClpStat = MagConv2ClpActPreExitClpr)  OR EDGENEG(p_bDIMagFixedClampSen))
						AND (p_eSelClampCtrlStatus = Done AND p_eSelClampCtrlStat = PneuActExt)
						AND (p_eSafetyBarStatus = Done AND p_eSafetyBarStat = PneuActExt)
						THEN
						eSelClampCtrl	:= PneuActIdle;
						eSafetyBarAct	:= PneuActIdle;
						eMagConv2ClpAct		:= MagConv2ClpActIdle;
						eGotoOpsStep		:= MagConvULStepMagExitedWait;

						bPaused	:= p_bStop OR p_bStep;
					END_IF
				MagConvULStepMagHalfExitMnl:
					sStepTxt	:= 'Magazine Conveyor HalfWay Exiting Magazine Manually';
					IF p_bProjLifTravMnlLoad = FALSE THEN

						eMagConv2ClpAct	:= MagConv2ClpActPreExitClpr1;
						eSelClampCtrl	:= PneuActExt;
						eSafetyBarAct	:= PneuActExt;
					ELSE
						eGotoOpsStep		:= MagConvULStepMagExitedWait; //no roller
					END_IF

					IF ((p_eMagConv2ClpStatus = Done AND p_eMagConv2ClpStat = MagConv2ClpActPreExitClpr1) OR EDGENEG(p_bDIMagFixedClampSen) )
						AND (p_eSelClampCtrlStatus = Done AND p_eSelClampCtrlStat = PneuActExt)
						AND (p_eSafetyBarStatus = Done AND p_eSafetyBarStat = PneuActExt)
						THEN
						eSelClampCtrl	:= PneuActIdle;
						eSafetyBarAct	:= PneuActIdle;
						eMagConv2ClpAct		:= MagConv2ClpActIdle;
						eGotoOpsStep		:= MagConvULStepMagExitedWait;

						bPaused	:= p_bStop OR p_bStep;
					END_IF
				MagConvULStepMagExitedWait:
					sStepTxt	:= 'Magazine Exited And Waiting For Remove';
					eAGVMagAct 	:= AGVMagActExit;
					IF bMagAutoEx THEN
						eDSSOTAct	:= SOTActRun;
					ELSE
						eDSSOTAct	:= SOTActIdle;
					END_IF

					bMagExitedWait	:= TRUE;

					fbEntSenOff(IN:= p_bLocalMagEntrySen = FALSE AND (NOT((p_bLocalBufferMagPresent OR p_bMag3OrientationChkSen1) AND p_bProjLifTravMnlLoad)));
					IF fbMagRemovedTm.Q OR fbEntSenOff.Q THEN
						bMagExitedWait	:= FALSE;
						ePrevExitStep 		:= MagConvULStepNA;
						iMagMESAcptCond 	:= 0;
						eGotoOpsStep	:= MagConvULStepMagUSComm;
						eDSSOTAct	:= SOTActIdle;

					ELSIF p_bNewMag = TRUE THEN
						bMagExitedWait	:= FALSE;
						eAGVMagAct 	:= AGVMagActIdle;
						ePrevExitStep 		:= MagConvULStepNA;
						iMagMESAcptCond 	:= 0;
						eGotoOpsStep	:= MagConvULStepMagEntMnl;
						eDSSOTAct			:= SOTActIdle;
					END_IF

					IF p_bAGVMagMcRunRdy = TRUE THEN
						eGotoOpsStep 	:= MagConvULStepMagFullExit;
					ELSIF p_bDSSOTConvStart= TRUE THEN
						eGotoOpsStep 	:= MagConvULStepMagFullExit;
					END_IF

					bPaused	:= p_bStop OR p_bStep;

			END_CASE

		END_IF

	END_IF

	bNewMagAllw	:= eOpsStep = MagConvULStepMagUSComm;

	bRlsMagAllw	:= ((eOpsStep = MagConvULStepMagCmp
					OR eOpsStep = MagConvULStepBffrUSComm
					OR eOpsStep = MagConvULStepMagFullDSComm
					OR eOpsStep = MagConvULStepBffrEntBrd
					OR (eOpsStep = MagConvULStepMagEntMESStdByChk AND fbReadRFIDTO.Q )
					OR (eOpsStep = MagConvULStepMagExtMESStdByChk AND fbWriteRFIDTO.Q) )
					);
	bEjectMESStep		:= 	eGotoOpsStep =  MagConvULStepMagExitMnl;
//	bEjectMESStep		:= 	eOpsStep = MagConvULStepMagEntMESStdByChk OR eOpsStep = MagConvULStepMagExtMESStdByChk	;
//	bEjectMagNotAllw	:= NOT((eOpsStep = MagConvULStepMagEntMESStdByChk AND fbReadRFIDTO.Q)
//						OR (eOpsStep = MagConvULStepMagExtMESStdByChk AND fbWriteRFIDTO.Q));

	Act_OpsInfo;

	//Operation State
	bOpsInitDone		 := eOpsStep > MagConvULStepInitMagConv;
	bStepMagExitedWait	 := eOpsStep = MagConvULStepMagExitedWait;
	bStepMagVerification := eOpsStep = MagConvULStepVerifyMag;
	bStepMagFullExit 	 := eOpsStep = MagConvULStepMagFullExit;
	bStepMagUSCom 		 := eOpsStep = MagConvULStepMagUSComm;

	bAGVComm3Rdy			:= (eOpsStep = MagConvULStepMagUSComm OR eOpsStep = MagConvULStepMagFullDSComm OR eOpsStep = MagConvULStepMagExitedWait
									OR eOpsStep = MagConvULStepMagEnt OR eOpsStep = MagConvULStepMagFullExit) AND p_bAGVMagMcRunRdy;
	bStepOpsMagAWDone 			:= eOpsStep = MagConvULStepMagAWMov AND eGotoOpsStep = MagConvULStepMagAWDisengage;
	bStepOpsPitchUpdated		:= eOpsStep = MagConvULStepMtyBffr AND eGotoOpsStep = MagConvULStepMagCmp;
	bStepPLCGrab				:= p_tyLocalBufferStat.bBffrMty AND EDGEPOS(p_bMagPresentSen);
END_ACTION
```

#### Act_OpsInfo.st
```iecst
ACTION Act_OpsInfo:

	//Reset
	udiStatus1	:= 0;

	IF p_bInfoEn = TRUE THEN

		//Magazine Not Present
		a_bMagAllwMagPresent[1]	:= p_bMagPresentSen1 OR p_bMagEntrySen1;
		a_bMagAllwMagPresent[2]	:= p_bMagPresentSen2 OR p_bMagEntrySen2;
		a_bMagAllwMagPresent[3]	:= p_bMagPresentSen3 OR p_bMagEntrySen3;

		FOR udi := 1 TO 3 DO
			IF pa_bMagDis[udi] = FALSE AND a_bMagAllwMagPresent[udi] = TRUE THEN
				EXIT;
			END_IF
		END_FOR

		IF udi = 4 THEN
			IF eOpsStep > MagConvULStepInitMagConv THEN
				udiStatus1	:= 10000;
			END_IF
		END_IF

		//Magazine Is Full
		a_tyMagAllwBffrStat[1]	:= p_tyBufferStat1;
		a_tyMagAllwBffrStat[2]	:= p_tyBufferStat2;
		a_tyMagAllwBffrStat[3]	:= p_tyBufferStat3;

		FOR udi := 1 TO 3 DO
			IF pa_bMagDis[udi] = FALSE AND a_bMagAllwMagPresent[udi] = TRUE AND a_tyMagAllwBffrStat[udi].bBffrFull = TRUE THEN
				udiStatus1	:= 10001 + (udi - 1);
				EXIT;
			END_IF
		END_FOR

		//Insert Good / Bad Magazine
		IF p_bConvInitDone = TRUE AND p_bConvHvBrd = TRUE THEN

			FOR udi := 1 TO 3 DO
				IF pa_bMagDis[udi] = FALSE AND pa_bMagRej[udi] = TRUE THEN
					EXIT;
				END_IF
			END_FOR

			IF udi < 4 THEN
				//Reject Mode
				IF p_bConvGdBrd = TRUE THEN
					//Good Board Exist
					FOR udi1 := 1 TO 3 DO
						IF pa_bMagDis[udi1] = FALSE AND a_bMagAllwMagPresent[udi1] = TRUE AND pa_bMagRej[udi1] = FALSE THEN
							EXIT;
						END_IF
					END_FOR

					IF udi1 = 4 THEN
						udiStatus1	:= 10004;
					END_IF

				ELSE
					//Bad Board Exist
					FOR udi1 := 1 TO 3 DO
						IF pa_bMagDis[udi1] = FALSE AND a_bMagAllwMagPresent[udi1] = TRUE AND pa_bMagRej[udi1] = TRUE THEN
							EXIT;
						END_IF
					END_FOR

					IF udi1 = 4 THEN
						udiStatus1	:= 10005;
					END_IF

				END_IF

			ELSE
				//Non-Reject Mode
				FOR udi1 := 1 TO 3 DO
					IF pa_bMagDis[udi1] = FALSE AND a_bMagAllwMagPresent[udi1] = TRUE THEN
						EXIT;
					END_IF
				END_FOR

				IF udi1 = 4 THEN
					udiStatus1	:= 10004;
				END_IF

			END_IF

		END_IF
END_IF

	//Magazine Verification Warning

	IF fbMagRemovedTm.Q OR bNewMagVerified THEN
		bNewMagVerifyStarted := FALSE;
	END_IF

	fbVerifyWarningDelay(IN:= bNewMagVerifyStarted AND bNewMagVerified = FALSE AND bStepMagVerification = FALSE);

	IF fbVerifyWarningDelay.Q AND p_tyBufferStat3.bBffrFull = FALSE THEN
		IF  (p_bMagAWCloseLimit OR  p_bMagAWOpenLimit) AND p_tyBufferStat3.bBffrMty THEN
			bLimitSenActivated := TRUE;
			udiStatus1	:= 10010;
		ELSIF bLimitSenActivated THEN
			udiStatus1	:= 10010;
		ELSIF bManualUnloadMag = FALSE THEN
			CASE p_bLinkMagRcpCurrRcpMagModel OF
				0: //CAB706.2
					IF bWrongHeight THEN
						udiStatus1	:= 10007;
					ELSIF p_bDIMagConvHeightSen = FALSE THEN
						bWrongHeight := TRUE;

					ELSIF bWrongWidth THEN
						udiStatus1	:= 10006;
					ELSIF p_bDIMagConvSelUnclampRS
						OR p_bDIMagConvCAB717Sen
						OR p_bDIMagConvSmallSen = FALSE
						THEN
						bWrongWidth := TRUE;

					END_IF

				1: //CAB716.2
					IF bWrongHeight THEN
						udiStatus1	:= 10007;
					ELSIF p_bDIMagConvHeightSen = TRUE THEN
						bWrongHeight := TRUE;

					ELSIF bWrongWidth THEN
						udiStatus1	:= 10006;
					ELSIF p_bDIMagConvSelUnclampRS
						OR p_bDIMagConvCAB717Sen
						OR p_bDIMagConvSmallSen = FALSE
						THEN
						bWrongWidth := TRUE;

					END_IF

				2: //CAB717.2
					IF bWrongHeight THEN
						udiStatus1	:= 10007;
					ELSIF p_bDIMagConvHeightSen THEN
						bWrongHeight := TRUE;

					ELSIF bWrongWidth THEN
						udiStatus1	:= 10006;
					ELSIF p_bDIMagConvSelUnclampRS = FALSE
						OR p_bDIMagConvCAB717Sen = FALSE
						OR p_bDIMagConvLargeSen
						THEN
						bWrongWidth := TRUE;

					END_IF

			END_CASE
		ELSIF bManualUnloadMag THEN
			udiStatus1	:= 10008;
		END_IF
	ELSIF udiStatus1 <> 10006
		AND udiStatus1 <> 10007
		AND p_tyBufferStat1.bBffrFull = FALSE
		AND bStepMagExitedWait
		AND p_bLocalMagEntrySen
		THEN
		udiStatus1	:= 10008;
		bManualUnloadMag := TRUE;

	ELSE
		bLimitSenActivated := FALSE;
		bWrongHeight := FALSE;
		bWrongWidth	:= FALSE;
	END_IF

	bIncorrectMagazineModel := udiStatus1 = 10006 OR udiStatus1 = 10007;

	//----------------------------Siemens MES -------------------------------------//
	IF (udiStatus1 = 0 OR udiStatus1 = 10008) AND (p_eCustomerReq = Siemens OR p_eCustomerReq = We_Fabricate)THEN
		IF eOpsStep = MagConvULStepMagEntMESStdByChk  THEN
			IF NOT(fbReadRFIDTO.Q) THEN //Reading RFID
				udiStatus1 := 10012;
			ELSE   //Reading RFID Time Out,Press Release Then Exit
				udiStatus1 := 10013;
			END_IF
		ELSIF eOpsStep = MagConvULStepMagExtMESStdByChk   THEN//
			IF NOT(fbWriteRFIDTO.Q) THEN
				udiStatus1 := 10014; //Writing RFID
			ELSE
				udiStatus1 := 10015; //Writing RFID , Press Release Mag
			END_IF
		ELSIF (eOpsStep = MagConvULStepMagFullDSComm OR eOpsStep = MagConvULStepMagExitMnl OR eOpsStep = MagConvULStepMagExitedWait)AND iMagMESAcptCond < 0  THEN
			udiStatus1 := 10016; //Wrong Magazine Position 3
		END_IF
	END_IF

END_ACTION
```

#### Act_OpsRst.st - Do Not Change!!!
```iecst
(** 2019-03-25 **)
ACTION Act_OpsRst:

	udiStatus1	:= 0;

	eBufferAct		:= BufferActIdle;
	eMagConv2ClpAct	:= MagConv2ClpActIdle;
	eUSSMEMAAct		:= SMEMAActIdle;
	eAGVMagAct		:= AGVMagActIdle;
	eSelClampCtrl	:= PneuActIdle;
	eSafetyBarAct	:= PneuActIdle;
	eMagAWEngageAct	:= PneuActIdle;
	eMagAWAct		:= MagAWActIdle;
	eDSSOTAct		:= SOTActIdle;
	eUSSOTAct		:= SOTActIdle;

	bNewMagVerified := FALSE;
	bNewMagVerifyStarted := FALSE;
	bReadRFID := FALSE;
	bWriteRFID := FALSE;
//	fbWriteRFIDTO(IN:= FALSE);

END_ACTION
```

### OpsLifMagUL.typ - Do Not Change!!!
```iecst
(*2018-12-11*)
(**)
(*Sequence*)

TYPE
	eLifMagULStep :
		(
		LifMagULStepNA,
		LifMagULStepMag1ConvInit,
		LifMagULStepMag2ConvInit,
		LifMagULStepInitLif,
		LifMagULStepMagCmp,
		LifMagULStepNxtLoadBffr,
		LifMagULStepLifMov,
		LifMagULStepBffrUSComm,
		LifMagULStepBffrEntBrd,
		LifMagULStepLoadBffr,
		LifMagULStepLifMovUnload,
		LifMagULStepUnload,
		LifMagULStepStandby,
		LiftMagConvInit,
		LiftMagConvIdle,
		LiftMagLifterLoad,
		LiftMagLifterUnload,
		LiftMagConvIN,
		LiftMagConvOUT
		);
	eLifMagULMagNxtLoad :
		(
		MagNxtLoadInvalid,
		MagNxtLoadMag1,
		MagNxtLoadMag2,
		MagNxtLoadMag3
		);
	eLifterConvStatus :
		(
		LifterNA := 0,
		LifterLoadPos := 1,
		LifterLoadRdyTrans := 2,
		LifterMagInProgress := 3,
		LifterUnloadPos := 4,
		LifterUnloadRdyTrans := 5
		);
END_TYPE
```

### OpsLifMagUL.var - Change By Project
```iecst
(*2019-03-25*)
(**)
(*Action & State & Status*)
(**)
(*Alarm*)
VAR
	p_OpsLifMagULAlmData : UDINT;
	p_OpsLifMagULAlmData1 : UDINT;
	p_OpsLifMagULAlmData2 : UDINT;
END_VAR
(**)
(*Output*)
VAR
	p_OpsLifMagULStepTxt : UDINT;
	p_OpsLifMagULStepTxt1 : UDINT;
	p_OpsLifMagULPaused : UDINT;
END_VAR
(**)
VAR
	p_OpsLifMagULLifterAct : UDINT;
	p_OpsLifMagULBufferAct1 : UDINT;
	p_OpsLifMagULBufferAct2 : UDINT;
	p_OpsLifMagULBufferAct3 : UDINT;
	p_OpsLifMagULUSSMEMAAct1 : UDINT;
	p_OpsLifMagULUSSMEMAAct2 : UDINT;
	p_OpsLifMagULUSSMEMAAct3 : UDINT;
END_VAR
(**)
VAR
	p_OpsLifMagULMagNxtLoad : UDINT;
	p_OpsLifMagULUnloading : UDINT;
	p_OpsLifMagULLiftMoving : UDINT;
	p_OpsLifMagULLifter2Act : UDINT;
	p_OpsLifMagULLifterConvAct : UDINT;
	p_OpsLifMagULLifterConv2Act : UDINT;
	p_OpsLifMagULStepInitDone1 : UDINT;
	p_OpsLifMagULStepInitDone2 : UDINT;
	p_OpsLifMagULStepEntMag1 : UDINT;
	p_OpsLifMagULStepExtMag1 : UDINT;
	p_OpsLifMagULStepEntMag2 : UDINT;
	p_OpsLifMagULStepExtMag2 : UDINT;
	p_OpsLifMagULStepIdle2 : UDINT;
END_VAR
```

### Program Logical/Operations/OpsLifMagUL (IEC) - 1.00.0 - 

#### InputRef.var
```iecst
(*2019-04-16*)
(**)
(*General*)
VAR
	p_udiRstErr : REFERENCE TO UDINT;
	p_bEn : REFERENCE TO BOOL;
	p_bDis : REFERENCE TO BOOL;
	p_bRun : REFERENCE TO BOOL;
	p_bStop : REFERENCE TO BOOL;
	p_bStep : REFERENCE TO BOOL;
END_VAR
(**)
(*Configuration*)
VAR
	p_sProgNm : REFERENCE TO STRING[15];
	p_bNtSettingsLoadDone : REFERENCE TO BOOL;
END_VAR
(**)
VAR
	pa_bMagDis : REFERENCE TO ARRAY[1..3] OF BOOL;
	pa_bMagRej : REFERENCE TO ARRAY[1..3] OF BOOL;
	p_bUnloadMag : REFERENCE TO BOOL;
	p_bUSAllow : REFERENCE TO BOOL;
	p_eNtParamProjMagBuffferActLoad : REFERENCE TO eLifMagULUpdateData;
END_VAR
(**)
VAR
	p_bConvInitDone : REFERENCE TO BOOL;
	p_bConvHvBrd : REFERENCE TO BOOL;
	p_bConvGdBrd : REFERENCE TO BOOL;
END_VAR
(**)
VAR
	p_tyBufferStat1 : REFERENCE TO tyBffrStat;
	p_tyBufferStat2 : REFERENCE TO tyBffrStat;
	p_tyBufferStat3 : REFERENCE TO tyBffrStat;
END_VAR
(**)
VAR
	p_bMagPresentSen1 : REFERENCE TO BOOL;
	p_bMagPresentSen2 : REFERENCE TO BOOL;
	p_bMagPresentSen3 : REFERENCE TO BOOL;
END_VAR
(**)
VAR
	p_bBufferMagPresent1 : REFERENCE TO BOOL;
	p_bBufferMagPresent2 : REFERENCE TO BOOL;
	p_bBufferMagPresent3 : REFERENCE TO BOOL;
END_VAR
(**)
VAR
	p_dtBufferMagPresentTm1 : REFERENCE TO DATE_AND_TIME;
	p_dtBufferMagPresentTm2 : REFERENCE TO DATE_AND_TIME;
	p_dtBufferMagPresentTm3 : REFERENCE TO DATE_AND_TIME;
END_VAR
(**)
VAR
	p_eLifterStat : REFERENCE TO eLifterAction;
	p_eLifterStatus : REFERENCE TO eFBStatus;
END_VAR
(**)
VAR
	p_eLifter2Stat : REFERENCE TO eLifterAction;
	p_eLifter2Status : REFERENCE TO eFBStatus;
END_VAR
(**)
VAR
	p_eLifterMagConvStat : REFERENCE TO eMagConvAction;
	p_eLifterMagConvStatus : REFERENCE TO eFBStatus;
	p_eLifterMagConv2Stat : REFERENCE TO eMagConvAction;
	p_eLifterMagConv2Status : REFERENCE TO eFBStatus;
END_VAR
(**)
VAR
	p_eInMagConvStat : REFERENCE TO eMagConvAction;
	p_eInMagConvStatus : REFERENCE TO eFBStatus;
	p_eOutMagConvStat : REFERENCE TO eMagConvAction;
	p_eOutMagConvStatus : REFERENCE TO eFBStatus;
	p_eInMagConv2Stat : REFERENCE TO eMagConvAction;
	p_eInMagConv2Status : REFERENCE TO eFBStatus;
	p_eOutMagConv2Stat : REFERENCE TO eMagConvAction;
	p_eOutMagConv2Status : REFERENCE TO eFBStatus;
END_VAR
(**)
VAR
	p_eBufferStat1 : REFERENCE TO eBufferAction;
	p_eBufferStatus1 : REFERENCE TO eFBStatus;
END_VAR
(**)
VAR
	p_eBufferStat2 : REFERENCE TO eBufferAction;
	p_eBufferStatus2 : REFERENCE TO eFBStatus;
END_VAR
(**)
VAR
	p_eBufferStat3 : REFERENCE TO eBufferAction;
	p_eBufferStatus3 : REFERENCE TO eFBStatus;
END_VAR
(**)
VAR
	p_eUSSMEMAStat1 : REFERENCE TO eSMEMAAction;
	p_eUSSMEMAStatus1 : REFERENCE TO eFBStatus;
	p_bUSSMEMATransporting1 : REFERENCE TO BOOL;
	p_bUSSMEMAConvStart1 : REFERENCE TO BOOL;
	p_bUSSMEMAConvStop1 : REFERENCE TO BOOL;
END_VAR
(**)
VAR
	p_eUSSMEMAStat2 : REFERENCE TO eSMEMAAction;
	p_eUSSMEMAStatus2 : REFERENCE TO eFBStatus;
	p_bUSSMEMATransporting2 : REFERENCE TO BOOL;
	p_bUSSMEMAConvStart2 : REFERENCE TO BOOL;
	p_bUSSMEMAConvStop2 : REFERENCE TO BOOL;
END_VAR
(**)
VAR
	p_eUSSMEMAStat3 : REFERENCE TO eSMEMAAction;
	p_eUSSMEMAStatus3 : REFERENCE TO eFBStatus;
	p_bUSSMEMATransporting3 : REFERENCE TO BOOL;
	p_bUSSMEMAConvStart3 : REFERENCE TO BOOL;
	p_bUSSMEMAConvStop3 : REFERENCE TO BOOL;
END_VAR
(*Shutter*)
VAR
	p_bDIInShutterOpenRS : REFERENCE TO BOOL;
	p_bDIInShutterCloseRS : REFERENCE TO BOOL;
	p_bDIOutShutterOpenRS : REFERENCE TO BOOL;
	p_bDIOutShutterCloseRS : REFERENCE TO BOOL;
	p_bDIPusherRetRS : REFERENCE TO BOOL;
	p_bMcParamMagFullBuzOff : REFERENCE TO BOOL;
END_VAR
(**)
VAR
	p_sProdRcpCurrRcp1Name : REFERENCE TO DINT;
	p_sProdRcpCurrRcp2Name : REFERENCE TO DINT;
END_VAR
(*MagConv*)
VAR
	p_usiMag1Rdy : REFERENCE TO eLifterConvStatus;
	p_usiMag2Rdy : REFERENCE TO eLifterConvStatus;
	p_bPresentMag1 : REFERENCE TO BOOL;
	p_bPresentMag2 : REFERENCE TO BOOL;
	p_bMagConvLanePrep : REFERENCE TO BOOL;
	p_bMagConvLane2Prep : REFERENCE TO BOOL;
	p_bNtParamProjLifter2Prep : REFERENCE TO BOOL;
	p_bOutShutterExtended : REFERENCE TO BOOL;
END_VAR
(**)
```

#### InputRef_Link.var
```iecst
(*2018-12-11*)
(**)
VAR
	p_bLinkFollower2USAllow : REFERENCE TO BOOL;
	p_bLinkDIInMagConvExtSen : REFERENCE TO BOOL;
	p_bLinkDIOutMagConvEntSen : REFERENCE TO BOOL;
	p_bLinkDIOutMagConvMidSen : REFERENCE TO BOOL;
	p_bLinkDIInMagConv2ExtSen : REFERENCE TO BOOL;
	p_bLinkDIOutMagConv2EntSen : REFERENCE TO BOOL;
	p_bLinkDIOutMagConv2MidSen : REFERENCE TO BOOL;
	p_bOpsOutMagConvStepInitDone : REFERENCE TO BOOL;
	p_bOpsOutMagConv2StepInitDone : REFERENCE TO BOOL;
	p_bLinkOpsMnlUnloadMag : REFERENCE TO BOOL;
	p_bLinkOpsOutMagConvStepWaitRmv : REFERENCE TO BOOL;
	p_bLinkOpsOutMagConv2StepWaitRmv : REFERENCE TO BOOL;
END_VAR
```

#### Local.var
```iecst
(*2019-04-16*)
(**)
(*Local Action, State & Status*)
VAR
	eStatus : eFBStatus := Idle;
	udiStatus : UDINT := 0;
	udiStatus1 : UDINT := 0;
	udiStatus2 : UDINT := 0;
END_VAR
(**)
(*Local Alarm*)
VAR
	tyAlmData : tyAlmDat;
	tyAlmData1 : tyAlmDat;
	tyAlmData2 : tyAlmDat;
	a_tyAlmText : ARRAY[10000..10099] OF tyAlmTxt := [(sAlmText:='Magazine Not Present'),(sAlmText:='Magazine 1 Is Full'),(sAlmText:='Magazine 2 Is Full'),(sAlmText:='Magazine 3 Is Full'),(sAlmText:='Please Insert Good Magazine'),(sAlmText:='Please Insert Bad Magazine'),2((sAlmText:='Last Magazine Is Almost Full')),(sAlmText:='All Magazines Full'),(sAlmText:='Please Insert Magazine'),90((0))];
END_VAR
(**)
(*Local Output*)
VAR
	sStepTxt : STRING[80];
	sStepTxt1 : STRING[80];
	bPaused : BOOL;
END_VAR
(**)
VAR
	eLifterAct : eLifterAction;
	eLifter2Act : eLifterAction;
	eBufferAct1 : eBufferAction;
	eBufferAct2 : eBufferAction;
	eBufferAct3 : eBufferAction;
	eUSSMEMAAct1 : eSMEMAAction;
	eUSSMEMAAct2 : eSMEMAAction;
	eUSSMEMAAct3 : eSMEMAAction;
END_VAR
(**)
VAR
	eMagNxtLoad : eLifMagULMagNxtLoad;
	bUnloading : BOOL;
	bLifterMoving : BOOL;
END_VAR
(**)
(*Local Input*)
VAR
	udiRstErr : UDINT := 0;
	bEn : BOOL := TRUE;
	bDis : BOOL := FALSE;
	bRun : BOOL;
	bStop : BOOL;
	bStep : BOOL;
	a_bMagDis : ARRAY[1..3] OF BOOL;
	a_bMagRej : ARRAY[1..3] OF BOOL;
	bUnloadMag : BOOL;
	bUSAllow : BOOL := TRUE;
	eMagBuffferActLoad : eLifMagULUpdateData;
	bConvInitDone : BOOL;
	bConvHvBrdAllwGo : BOOL;
	bConvHvBrd : BOOL;
	bConvGdBrd : BOOL;
	tyBufferStat1 : tyBffrStat;
	tyBufferStat2 : tyBffrStat;
	tyBufferStat3 : tyBffrStat;
	bMagPresentSen1 : BOOL;
	bMagPresentSen2 : BOOL;
	bMagPresentSen3 : BOOL;
	bBufferMagPresent1 : BOOL;
	bBufferMagPresent2 : BOOL;
	bBufferMagPresent3 : BOOL;
	dtBufferMagPresentTm1 : DATE_AND_TIME;
	dtBufferMagPresentTm2 : DATE_AND_TIME;
	dtBufferMagPresentTm3 : DATE_AND_TIME;
	eLifterStat : eLifterAction;
	eLifterStatus : eFBStatus;
	eLifter2Stat : eLifterAction;
	eLifter2Status : eFBStatus;
	eBufferStat1 : eBufferAction;
	eBufferStatus1 : eFBStatus;
	eBufferStat2 : eBufferAction;
	eBufferStatus2 : eFBStatus;
	eBufferStat3 : eBufferAction;
	eBufferStatus3 : eFBStatus;
	eUSSMEMAStat1 : eSMEMAAction;
	eUSSMEMAStatus1 : eFBStatus;
	bUSSMEMATransporting1 : BOOL;
	bUSSMEMAConvStart1 : BOOL;
	bUSSMEMAConvStop1 : BOOL;
	eUSSMEMAStat2 : eSMEMAAction;
	eUSSMEMAStatus2 : eFBStatus;
	bUSSMEMATransporting2 : BOOL;
	bUSSMEMAConvStart2 : BOOL;
	bUSSMEMAConvStop2 : BOOL;
	eUSSMEMAStat3 : eSMEMAAction;
	eUSSMEMAStatus3 : eFBStatus;
	bUSSMEMATransporting3 : BOOL;
	bUSSMEMAConvStart3 : BOOL;
	bUSSMEMAConvStop3 : BOOL;
	sProgNm : STRING[15] := 'Ops LifMagUL';
	bNtSettingsLoadDone : BOOL := TRUE;
END_VAR
(**)
(*Local*)
VAR
	bRstErr : BOOL;
	udiRstErrOld : UDINT;
	bInitDone : BOOL;
	bInitialDone : BOOL;
	eOpsStep : eLifMagULStep := LifMagULStepNA;
	eGotoOpsStep : eLifMagULStep := LifMagULStepInitLif;
	eOpsStep1 : eLifMagULStep := LifMagULStepNA;
	eGotoOpsStep1 : eLifMagULStep := LiftMagConvInit;
	eOpsStep2 : eLifMagULStep := LifMagULStepNA;
	eGotoOpsStep2 : eLifMagULStep := LiftMagConvInit;
	udi : UDINT;
	udi1 : UDINT;
	udiCount : UDINT;
	udiCmpTm : UDINT;
	udiMagAllwGo : UDINT;
	bMagNxtUnloadGd : BOOL;
	a_tyMagAllwBffrStat : ARRAY[1..3] OF tyBffrStat;
	a_bMagAllwMagPresent : ARRAY[1..3] OF BOOL;
	a_udiMagAllwMagPresentTm : ARRAY[1..3] OF UDINT;
	a_udiMagAllwPriority : ARRAY[1..3] OF UDINT;
	a_udiMagAllwSum : ARRAY[1..3] OF UDINT;
	p_tyLocalBufferStat : REFERENCE TO tyBffrStat;
	p_bLocalBufferMagPresent : REFERENCE TO BOOL;
	p_dtLocalBufferMagPresentTm : REFERENCE TO DATE_AND_TIME;
	p_eLocalBufferAct : REFERENCE TO eBufferAction;
	p_eLocalBufferStat : REFERENCE TO eBufferAction;
	p_eLocalBufferStatus : REFERENCE TO eFBStatus;
	p_eLocalUSSMEMAAct : REFERENCE TO eSMEMAAction;
	p_eLocalUSSMEMAStat : REFERENCE TO eSMEMAAction;
	p_eLocalUSSMEMAStatus : REFERENCE TO eFBStatus;
	p_bLocalUSSMEMATransporting : REFERENCE TO BOOL;
	p_bLocalUSSMEMAConvStart : REFERENCE TO BOOL;
	p_bLocalUSSMEMAConvStop : REFERENCE TO BOOL;
END_VAR
(*local LiftConv*)
VAR
	bLocalMag1InPos : BOOL;
	bLocalMag2InPos : BOOL;
	bLift2Move : BOOL;
	usiMag1Rdy : eLifterConvStatus;
	usiMag2Rdy : eLifterConvStatus;
	bStepEntMag1 : BOOL;
	bStepExtMag1 : BOOL;
	bStepEntMag2 : BOOL;
	bStepExtMag2 : BOOL;
	bStepInitDone1 : BOOL;
	bStepInitDone2 : BOOL;
	bPresentMag1 : BOOL;
	bPresentMag2 : BOOL;
	bStepLiftMagIdle2 : BOOL;
	bMagConvLanePrep : BOOL;
	bStepEntBoard : BOOL;
	bMagSetFullExit : BOOL;
	bMagSetFullExit2 : BOOL;
	udiModuleNum : UDINT := 6091;
END_VAR
```

#### Act_Alarm.st
```iecst
(** 2019-03-25 **)
ACTION Act_Alarm:

	//Error
	IF EDGEPOS(eStatus = Error) THEN

		tyAlmData.sProgNm		:= p_sProgNm;
		tyAlmData.udiCode		:= udiStatus;
		tyAlmData.eSeverity		:= AlmSeverityError;
		tyAlmData.udiRunTime	:= tyAlmData.udiRunTime + 1;
		tyAlmData.bAlm			:= TRUE;
		tyAlmData.udiModuleNum  := udiModuleNum;
		g_sOpsLifMagULProgNm		:= p_sProgNm;

		//Get Error Message
		IF tyAlmData.udiCode < 10000 OR tyAlmData.udiCode > 10099 THEN
			tyAlmData.sAlmMsg	:= 'Unknown';
			tyAlmData.sRcyMsg	:= 'Unknown';
		ELSE
			tyAlmData.sAlmMsg	:= a_tyAlmText[tyAlmData.udiCode].sAlmText;
			tyAlmData.sRcyMsg	:= a_tyAlmText[tyAlmData.udiCode].sRcyText;
		END_IF

	ELSIF bRstErr AND (tyAlmData.udiCode <> 0) THEN

		tyAlmData.udiCode		:= 0;
		tyAlmData.eSeverity		:= AlmSeverityNA;
		tyAlmData.sAlmMsg		:= '';
		tyAlmData.sRcyMsg		:= '';
		tyAlmData.bAlm			:= FALSE;
	END_IF

END_ACTION
```

#### Act_AlarmInfo1.st
```iecst
(** 2019-03-25 **)
ACTION Act_AlarmInfo1:

	//Info
	tyAlmData1.sProgNm		:= p_sProgNm;
	tyAlmData1.udiCode		:= udiStatus1;
	tyAlmData1.eSeverity	:= AlmSeverityInfo;
	tyAlmData1.udiRunTime	:= tyAlmData1.udiRunTime + 1;

	//Get Info Message
	IF tyAlmData1.udiCode < 10000 OR tyAlmData1.udiCode > 10099 THEN
		tyAlmData1.sAlmMsg	:= 'Unknown';
		tyAlmData1.sRcyMsg	:= 'Unknown';
	ELSE
		tyAlmData1.sAlmMsg	:= a_tyAlmText[tyAlmData1.udiCode].sAlmText;
		tyAlmData1.sRcyMsg	:= a_tyAlmText[tyAlmData1.udiCode].sRcyText;
	END_IF

END_ACTION
```

#### Act_InitGlobal.st
```iecst
(** 2019-04-16 **)
ACTION Act_InitGlobal:

	(* Always Change If Project Change *)

	//Pass Data To Link
	p_bLinkDIInMagConvExtSen ACCESS p_DIInMagConvExtSen;
	p_bLinkDIOutMagConvEntSen ACCESS p_DIOutMagConvEntSen;
	p_bLinkDIOutMagConvMidSen ACCESS p_DIOutMagConvMidSen;

	p_bLinkDIInMagConv2ExtSen ACCESS p_DIInMagConv2ExtSen;
	p_bLinkDIOutMagConv2EntSen ACCESS p_DIOutMagConv2EntSen;
	p_bLinkDIOutMagConv2MidSen ACCESS p_DIOutMagConv2MidSen;

	p_bOpsOutMagConvStepInitDone ACCESS p_OpsOutMagConvStepInitDone;
	p_bOpsOutMagConv2StepInitDone ACCESS p_OpsOutMagConv2StepInitDone;

	p_bLinkOpsMnlUnloadMag ACCESS p_UIOpsMnlUnloadMag; //no use
	p_bLinkOpsOutMagConvStepWaitRmv ACCESS p_OpsOutMagConvStepWaitToRmvMag;
	p_bLinkOpsOutMagConv2StepWaitRmv ACCESS p_OpsOutMagConv2StepWaitToRmvMag;

	//Pass Data To Internal Use
	p_udiRstErr ACCESS p_RstErrReset;
	p_bRun ACCESS p_OpsRun;
	p_bStop ACCESS p_OpsStop;
	p_bStep ACCESS p_OpsStep;

	p_sProgNm ACCESS p_NtParamOpsMagUL1ProgNm;
	p_bNtSettingsLoadDone ACCESS p_StartupNtSettingsLoadDone;

	pa_bMagDis ACCESS p_OpsTravLifULMagDis;
	pa_bMagRej ACCESS p_OpsTravLifULMagRej;
	p_bUnloadMag ACCESS p_UIUnloadMag;
	p_bLinkFollower2USAllow ACCESS p_Follower2USAllow;
	p_eNtParamProjMagBuffferActLoad	ACCESS p_NtParamProjMagBuffferActLoad;

	p_bConvInitDone ACCESS p_OpsTravLifULInitDone;
	p_bConvHvBrd ACCESS p_PshrConvHvBrd;
	p_bConvGdBrd ACCESS p_PshrConvGdBrd;

	p_tyBufferStat1 ACCESS p_Buffer1BffrStat;
	p_tyBufferStat2 ACCESS p_Buffer2BffrStat;
	p_tyBufferStat3 ACCESS p_Buffer3BffrStat;

	p_bMagPresentSen1 ACCESS p_DIMagPresentSen1; // == lifterlimitSW ,no need assign again
	p_bMagPresentSen2 ACCESS p_DIMagPresentSen2; // == lifterlimitSW2,no need assign again
	p_bMagPresentSen3 ACCESS p_DIMagPresentSen3;

	p_bBufferMagPresent1 ACCESS p_Buffer1MagPresent;
	p_bBufferMagPresent2 ACCESS p_Buffer2MagPresent;
	p_bBufferMagPresent3 ACCESS p_Buffer3MagPresent;

	p_dtBufferMagPresentTm1 ACCESS p_Buffer1MagPresentTm;
	p_dtBufferMagPresentTm2 ACCESS p_Buffer2MagPresentTm;
	p_dtBufferMagPresentTm3 ACCESS p_Buffer3MagPresentTm;

	p_eLifterStat ACCESS p_LifterBtmStat;
	p_eLifterStatus ACCESS p_LifterBtmStatus;

	p_eBufferStat1 ACCESS p_Buffer1Stat;
	p_eBufferStatus1 ACCESS p_Buffer1Status;

	p_eBufferStat2 ACCESS p_Buffer2Stat;
	p_eBufferStatus2 ACCESS p_Buffer2Status;

	p_eBufferStat3 ACCESS p_Buffer3Stat;
	p_eBufferStatus3 ACCESS p_Buffer3Status;

	p_eUSSMEMAStat1 ACCESS p_USSMEMA1Stat;
	p_eUSSMEMAStatus1 ACCESS p_USSMEMA1Status;
	p_bUSSMEMATransporting1 ACCESS p_USSMEMA1Transporting;
	p_bUSSMEMAConvStart1 ACCESS p_USSMEMA1ConvStart;
	p_bUSSMEMAConvStop1 ACCESS p_USSMEMA1ConvStop;

	p_eUSSMEMAStat2 ACCESS p_USSMEMA2Stat;
	p_eUSSMEMAStatus2 ACCESS p_USSMEMA2Status;
	p_bUSSMEMATransporting2 ACCESS p_USSMEMA2Transporting;
	p_bUSSMEMAConvStart2 ACCESS p_USSMEMA2ConvStart;
	p_bUSSMEMAConvStop2 ACCESS p_USSMEMA2ConvStop;

	p_eUSSMEMAStat3 ACCESS p_USSMEMA3Stat;
	p_eUSSMEMAStatus3 ACCESS p_USSMEMA3Status;
	p_bUSSMEMATransporting3 ACCESS p_USSMEMA3Transporting;
	p_bUSSMEMAConvStart3 ACCESS p_USSMEMA3ConvStart;
	p_bUSSMEMAConvStop3 ACCESS p_USSMEMA3ConvStop;

	p_bDIInShutterOpenRS ACCESS p_DIInShutterOpenRS;
	p_bDIInShutterCloseRS ACCESS p_DIInShutterCloseRS;
	p_bDIOutShutterOpenRS ACCESS p_DIOutShutterOpenRS;
	p_bDIOutShutterCloseRS ACCESS p_DIOutShutterCloseRS;

	p_bDIPusherRetRS ACCESS p_DIPusherRetRS;

	p_sProdRcpCurrRcp1Name ACCESS p_ProdRcpCurrRcp1Nm;
	p_sProdRcpCurrRcp2Name ACCESS p_ProdRcpCurrRcp2Nm;

	//Lifter Conv
	p_eLifter2Stat ACCESS p_Lifter2Stat;
	p_eLifter2Status ACCESS p_Lifter2Status;
	p_eLifterMagConvStat ACCESS p_LifterMagConvStat;
	p_eLifterMagConvStatus ACCESS p_LifterMagConvStatus;
	p_eLifterMagConv2Stat ACCESS p_LifterMagConv2Stat;
	p_eLifterMagConv2Status ACCESS p_LifterMagConv2Status;
	//IN out mag conv
	p_eInMagConvStat ACCESS p_InMagConvStat;
	p_eInMagConvStatus ACCESS p_InMagConvStatus;
	p_eOutMagConvStat ACCESS p_OutMagConvStat;
	p_eOutMagConvStatus ACCESS p_OutMagConvStatus;
	p_eInMagConv2Stat ACCESS p_InMagConv2Stat;
	p_eInMagConv2Status ACCESS p_InMagConv2Stat;
	p_eOutMagConv2Stat ACCESS p_OutMagConv2Stat;
	p_eOutMagConv2Status ACCESS p_OutMagConv2Stat;

	p_bMagConvLanePrep ACCESS p_NtParamProjMagConvLane1Prep;
	p_bMagConvLane2Prep ACCESS p_NtParamProjMagConvLane2Prep;
	p_bNtParamProjLifter2Prep ACCESS p_NtParamProjLifter2Prep;
	p_bOutShutterExtended ACCESS p_Pneu2SenOutShutterExtended;

	p_bEn ACCESS p_NtParamProjLifterMagPlatform; // Added

	(* Always Change If Project Change *)

END_ACTION
```

#### Act_InitLocal.st
```iecst
(** 2019-04-16 **)
ACTION Act_InitLocal:

	//Input Reference Link To Local Variable
	p_udiRstErr ACCESS ADR(udiRstErr);
	p_bEn ACCESS ADR(bEn);
	p_bDis ACCESS ADR(bDis);
	p_bRun ACCESS ADR(bRun);
	p_bStop ACCESS ADR(bStop);
	p_bStep ACCESS ADR(bStep);

	p_sProgNm ACCESS ADR(sProgNm);
	p_bNtSettingsLoadDone ACCESS ADR(bNtSettingsLoadDone);

	pa_bMagDis ACCESS ADR(a_bMagDis);
	pa_bMagRej ACCESS ADR(a_bMagRej);
	p_bUnloadMag ACCESS ADR(bUnloadMag);
	p_bUSAllow ACCESS ADR(bUSAllow);
	p_eNtParamProjMagBuffferActLoad	ACCESS ADR(eMagBuffferActLoad);

	p_bConvInitDone ACCESS ADR(bConvInitDone);
	p_bConvHvBrd ACCESS ADR(bConvHvBrd);
	p_bConvGdBrd ACCESS ADR(bConvGdBrd);

	p_tyBufferStat1 ACCESS ADR(tyBufferStat1);
	p_tyBufferStat2 ACCESS ADR(tyBufferStat2);
	p_tyBufferStat3 ACCESS ADR(tyBufferStat3);

	p_bMagPresentSen1 ACCESS ADR(bMagPresentSen1);
	p_bMagPresentSen2 ACCESS ADR(bMagPresentSen2);
	p_bMagPresentSen3 ACCESS ADR(bMagPresentSen3);

	p_bBufferMagPresent1 ACCESS ADR(bBufferMagPresent1);
	p_bBufferMagPresent2 ACCESS ADR(bBufferMagPresent2);
	p_bBufferMagPresent3 ACCESS ADR(bBufferMagPresent3);

	p_dtBufferMagPresentTm1 ACCESS ADR(dtBufferMagPresentTm1);
	p_dtBufferMagPresentTm2 ACCESS ADR(dtBufferMagPresentTm2);
	p_dtBufferMagPresentTm3 ACCESS ADR(dtBufferMagPresentTm3);

	p_eLifterStat ACCESS ADR(eLifterStat);
	p_eLifterStatus ACCESS ADR(eLifterStatus);

	p_eBufferStat1 ACCESS ADR(eBufferStat1);
	p_eBufferStatus1 ACCESS ADR(eBufferStatus1);

	p_eBufferStat2 ACCESS ADR(eBufferStat2);
	p_eBufferStatus2 ACCESS ADR(eBufferStatus2);

	p_eBufferStat3 ACCESS ADR(eBufferStat3);
	p_eBufferStatus3 ACCESS ADR(eBufferStatus3);

	p_eUSSMEMAStat1 ACCESS ADR(eUSSMEMAStat1);
	p_eUSSMEMAStatus1 ACCESS ADR(eUSSMEMAStatus1);
	p_bUSSMEMATransporting1 ACCESS ADR(bUSSMEMATransporting1);
	p_bUSSMEMAConvStart1 ACCESS ADR(bUSSMEMAConvStart1);
	p_bUSSMEMAConvStop1 ACCESS ADR(bUSSMEMAConvStop1);

	p_eUSSMEMAStat2 ACCESS ADR(eUSSMEMAStat2);
	p_eUSSMEMAStatus2 ACCESS ADR(eUSSMEMAStatus2);
	p_bUSSMEMATransporting2 ACCESS ADR(bUSSMEMATransporting2);
	p_bUSSMEMAConvStart2 ACCESS ADR(bUSSMEMAConvStart2);
	p_bUSSMEMAConvStop2 ACCESS ADR(bUSSMEMAConvStop2);

	p_eUSSMEMAStat3 ACCESS ADR(eUSSMEMAStat3);
	p_eUSSMEMAStatus3 ACCESS ADR(eUSSMEMAStatus3);
	p_bUSSMEMATransporting3 ACCESS ADR(bUSSMEMATransporting3);
	p_bUSSMEMAConvStart3 ACCESS ADR(bUSSMEMAConvStart3);
	p_bUSSMEMAConvStop3 ACCESS ADR(bUSSMEMAConvStop3);

	//Lifter Conv
	p_eLifter2Stat ACCESS ADR(eLifter2Stat);
	p_eLifter2Status ACCESS ADR(eLifter2Status);
	p_eLifterMagConvStat ACCESS ADR(eLifterMagConvStat);
	p_eLifterMagConvStatus ACCESS ADR(eLifterMagConvStatus);
	p_eLifterMagConv2Stat ACCESS ADR(eLifterMagConv2Stat);
	p_eLifterMagConv2Status ACCESS ADR(eLifterMagConv2Status);
	//IN out mag conv
	p_eInMagConvStat ACCESS ADR(eInMagConvStat);
	p_eInMagConvStatus ACCESS ADR(eInMagConvStatus);
	p_eOutMagConvStat ACCESS ADR(eOutMagConvStat);
	p_eOutMagConvStatus ACCESS ADR(eOutMagConvStatus);
	p_eInMagConv2Stat ACCESS ADR(eInMagConv2Stat);
	p_eInMagConv2Status ACCESS ADR(eInMagConv2Status);
	p_eOutMagConv2Stat ACCESS ADR(eOutMagConv2Stat);
	p_eOutMagConv2Status ACCESS ADR(eOutMagConv2Status);

	p_usiMag1Rdy ACCESS ADR(usiMag1Rdy);
	p_usiMag2Rdy ACCESS ADR(usiMag2Rdy);
	p_bPresentMag1 ACCESS ADR(bPresentMag1);
	p_bPresentMag2 ACCESS ADR(bPresentMag2);

	p_bMagConvLanePrep ACCESS ADR(bMagConvLanePrep);
END_ACTION
```

#### Act_Link.st
```iecst
(** 2018-12-11 **)
ACTION Act_Link:

	//Upstream Allowed

	p_bUSAllow	:=  p_bLinkFollower2USAllow AND p_sProdRcpCurrRcp1Name = p_sProdRcpCurrRcp2Name;// OR p_bLinkTravULUSWidthChkBrdExist ;

	//Lifter status
	IF p_bMagConvLanePrep AND p_bMagConvLane2Prep THEN
		IF usiMag1Rdy = LifterLoadPos AND p_bLinkDIInMagConvExtSen THEN
			usiMag1Rdy := LifterLoadRdyTrans;
		ELSIF usiMag1Rdy = LifterUnloadPos AND p_bLinkDIOutMagConvEntSen = FALSE AND p_bLinkDIOutMagConvMidSen = FALSE
			AND p_bOpsOutMagConvStepInitDone AND p_bLinkOpsOutMagConvStepWaitRmv = FALSE THEN
			usiMag1Rdy := LifterUnloadRdyTrans;
		END_IF

		IF p_usiMag2Rdy = LifterLoadPos AND p_bLinkDIInMagConv2ExtSen THEN
			p_usiMag2Rdy := LifterLoadRdyTrans;
		ELSIF p_usiMag2Rdy = LifterUnloadPos AND p_bLinkDIOutMagConv2EntSen = FALSE AND p_bLinkDIOutMagConv2MidSen = FALSE
			AND p_bOpsOutMagConv2StepInitDone AND p_bLinkOpsOutMagConv2StepWaitRmv = FALSE THEN
			p_usiMag2Rdy := LifterUnloadRdyTrans;
		END_IF
	END_IF
END_ACTION
```

#### Cyclic.st
```iecst
(** 2019-03-22 **)
PROGRAM _CYCLIC

	IF bInitDone = FALSE THEN
		bInitDone	:= TRUE;

		Act_InitLocal;
		Act_InitGlobal;

	ELSIF bInitialDone = FALSE THEN
		IF p_bNtSettingsLoadDone = TRUE THEN
			bInitialDone	:= TRUE;

			Act_Initial;
		END_IF

	ELSE

		Act_RstErr;
		Act_LinkEn;
		Act_Link;
		Act_Background;
		Act_Alarm;
		Act_AlarmInfo1;

	END_IF

END_PROGRAM
```

#### Init.st
```iecst
(** 2019-03-25 **)
PROGRAM _INIT

	(* Always Change If Project Change *)

	//Pass Address To Global Address For External Use
	//Action, State & Status

	//Alarm
	p_OpsLifMagULAlmData	:= ADR(tyAlmData);
	p_OpsLifMagULAlmData1	:= ADR(tyAlmData1);
	p_OpsLifMagULAlmData2	:= ADR(tyAlmData2);
	//Output
	p_OpsLifMagULStepTxt	:= ADR(sStepTxt);
	p_OpsLifMagULStepTxt1	:= ADR(sStepTxt1);
	p_OpsLifMagULPaused		:= ADR(bPaused);

	p_OpsLifMagULLifterAct		:= ADR(eLifterAct);
	p_OpsLifMagULBufferAct1		:= ADR(eBufferAct1);
	p_OpsLifMagULBufferAct2		:= ADR(eBufferAct2);
	p_OpsLifMagULBufferAct3		:= ADR(eBufferAct3);
	p_OpsLifMagULUSSMEMAAct1	:= ADR(eUSSMEMAAct1);
	p_OpsLifMagULUSSMEMAAct2	:= ADR(eUSSMEMAAct2);
	p_OpsLifMagULUSSMEMAAct3	:= ADR(eUSSMEMAAct3);

	p_OpsLifMagULMagNxtLoad	:= ADR(eMagNxtLoad);
	p_OpsLifMagULUnloading	:= ADR(bUnloading);
	p_OpsLifMagULLiftMoving	:= ADR(bLifterMoving);

	p_OpsLifMagULLifter2Act		:= ADR(eLifter2Act);
	p_OpsLifMagULLifterConvAct		:= ADR(eLifterConvAct);
	p_OpsLifMagULLifterConv2Act		:= ADR(eLifterConv2Act);

	p_OpsLifMagULStepInitDone1			:= ADR(bStepInitDone1);
	p_OpsLifMagULStepInitDone2			:= ADR(bStepInitDone2);
	p_OpsLifMagULStepEntMag1			:= ADR(bStepEntMag1);
	p_OpsLifMagULStepExtMag1			:= ADR(bStepExtMag1);
	p_OpsLifMagULStepEntMag2			:= ADR(bStepEntMag2);
	p_OpsLifMagULStepExtMag2			:= ADR(bStepExtMag2);
	p_OpsLifMagULStepIdle2				:= ADR(bStepLiftMagIdle2);

	(* Always Change If Project Change *)

END_PROGRAM
```

#### Act_OpsInitial.st - Do Not Change!!!
```iecst
(** 2019-01-16 **)
ACTION Act_OpsInitial:

	eOpsStep		:= LifMagULStepNA;
	eGotoOpsStep	:= LifMagULStepInitLif;
	eOpsStep1		:= LifMagULStepNA;
	eGotoOpsStep1	:= LiftMagConvInit;
	eOpsStep2		:= LifMagULStepNA;
	eGotoOpsStep2	:= LiftMagConvInit;

END_ACTION
```

#### Act_OpsRun.st
```iecst
(** 2019-04-16 **)
ACTION Act_OpsRun:

	(*Unloader's Lifter Magazine Layout*)
	(*
		Direction: -->> Left To Right -->>

	                      +----------+
	                      |          |
	                      |          |
	     (Lif=PosCSlt) US3|          |
	               [Mag 3]|          |
	                      |          |
	     (Lif=PosBSlt) US2|          |
	               [Mag 2]|          |
	                      |          |
	     (Lif=PosASlt) US1|          |
	               [Mag 1]|          |
	                      | Unloader |
	                      +----------+

		Note: Program Action Called For Lifter As Shown Above
		      Setup Lifter Program Parameters Accordingly

	For 2 lane magconv
	-eGotoOpsStep, eGotoOpsStep1 will consider lane 1; eGotoOpsStep2,eGotoOpsStep3 consider lane 2
	i. Lifter move position D,E ; Load, Unload pos
	ii. Lifter 2 move position G,H ; Load, Unload pos
	*)

	IF eGotoOpsStep <> eOpsStep THEN

		CASE eGotoOpsStep OF
			LifMagULStepInitLif:
				IF NOT(p_bMagConvLanePrep) OR
					(p_bMagConvLanePrep  AND eOpsStep1 > LiftMagConvInit) THEN
					eOpsStep	:= eGotoOpsStep;
				END_IF
			ELSE
				eOpsStep	:= eGotoOpsStep;

		END_CASE

	END_IF

	IF eOpsStep = eGotoOpsStep THEN

		IF bPaused = FALSE THEN

			CASE eOpsStep OF

				LifMagULStepInitLif:
					sStepTxt	:= 'Initializing Lifter';
					IF p_bDIOutShutterCloseRS = TRUE THEN
						eLifterAct	:= LifterActFullHm;
					END_IF

					IF p_eLifterStatus = Done AND p_eLifterStat = LifterActFullHm THEN
						eLifterAct	:= LifterActIdle;
						eGotoOpsStep	:= LifMagULStepMagCmp;
						bPaused	:= p_bStop OR p_bStep;
					END_IF

				LifMagULStepMagCmp:
					sStepTxt	:= 'Comparing Magazine';

					a_tyMagAllwBffrStat[1]	:= p_tyBufferStat1;
					a_tyMagAllwBffrStat[2]	:= p_tyBufferStat2;
					a_tyMagAllwBffrStat[3]	:= p_tyBufferStat3;

					a_bMagAllwMagPresent[1]	:= p_bBufferMagPresent1;
					a_bMagAllwMagPresent[2]	:= p_bBufferMagPresent2;
					a_bMagAllwMagPresent[3]	:= p_bBufferMagPresent3;

					a_udiMagAllwMagPresentTm[1]	:= DT_TO_UDINT(p_dtBufferMagPresentTm1);
					a_udiMagAllwMagPresentTm[2]	:= DT_TO_UDINT(p_dtBufferMagPresentTm2);
					a_udiMagAllwMagPresentTm[3]	:= DT_TO_UDINT(p_dtBufferMagPresentTm3);

					//Sorting Priority
					memset(ADR(a_udiMagAllwPriority), 0, SIZEOF(a_udiMagAllwPriority));

					FOR udi := 1 TO 3 DO
						udiCount	:= 3;
						udiCmpTm	:= a_udiMagAllwMagPresentTm[udi];

						FOR udi1 := 1 TO 3 DO
							IF a_udiMagAllwMagPresentTm[udi1] > udiCmpTm THEN
								udiCount	:= udiCount - 1;
							END_IF
						END_FOR

						a_udiMagAllwPriority[udi]	:= udiCount;
					END_FOR

					FOR udi := 3 TO 1 BY -1 DO
						FOR udi1 := 3 TO 1 BY -1 DO
							IF (udi <> udi1) AND (a_udiMagAllwPriority[udi] = a_udiMagAllwPriority[udi1]) THEN
								a_udiMagAllwPriority[udi1]	:= a_udiMagAllwPriority[udi1] - 1;
							END_IF
						END_FOR
					END_FOR

					//Checking Buffer Status
					memset(ADR(a_udiMagAllwSum), 0, SIZEOF(a_udiMagAllwSum));

					FOR udi := 1 TO 3 DO
						//Priority
						a_udiMagAllwSum[udi]	:= a_udiMagAllwSum[udi] + a_udiMagAllwPriority[udi];
						//Enable
						IF pa_bMagDis[udi] = FALSE THEN
							a_udiMagAllwSum[udi]	:= a_udiMagAllwSum[udi] + 1000;
						END_IF
						//Magazine Present
						IF a_bMagAllwMagPresent[udi] = TRUE THEN
							a_udiMagAllwSum[udi]	:= a_udiMagAllwSum[udi] + 1000;
						END_IF
						//Magazine Empty
						IF a_tyMagAllwBffrStat[udi].bBffrMty = TRUE THEN
							a_udiMagAllwSum[udi]	:= a_udiMagAllwSum[udi] + 2500;
						END_IF
						//Magazine Available
						IF a_tyMagAllwBffrStat[udi].bBffrFull = FALSE AND a_tyMagAllwBffrStat[udi].bBffrMty = FALSE THEN
							a_udiMagAllwSum[udi]	:= a_udiMagAllwSum[udi] + 3000;
						END_IF
						//Magazine Reject
						IF pa_bMagRej[udi] = TRUE THEN
							a_udiMagAllwSum[udi]	:= a_udiMagAllwSum[udi] + 6000;
						END_IF

					END_FOR

					IF pa_bMagRej[1] = FALSE
						AND pa_bMagRej[2] = FALSE
						AND pa_bMagRej[3] = FALSE
					THEN
						bConvHvBrdAllwGo := p_bConvHvBrd;
					ELSE
						bConvHvBrdAllwGo := FALSE;
					END_IF

					udiMagAllwGo	:= 99;

					FOR udi := 1 TO 3 DO

						IF (a_udiMagAllwSum[udi] >= 5000 AND a_udiMagAllwSum[udi] < 6000 AND (p_bConvGdBrd = TRUE OR bConvHvBrdAllwGo))	//Enable + Magazine Present + Magazine Available
							OR (a_udiMagAllwSum[udi] >= 11000 AND p_bConvGdBrd = FALSE) THEN						//Reject + Enable + Magazine Present + Magazine Available

							IF udiMagAllwGo <> 99 THEN
								//Priority
								IF a_udiMagAllwSum[udi] < a_udiMagAllwSum[udiMagAllwGo] THEN
									udiMagAllwGo	:= udi;
								END_IF
							ELSE
								udiMagAllwGo	:= udi;
							END_IF

						END_IF

					END_FOR

					IF udiMagAllwGo = 99 THEN

						FOR udi := 1 TO 3 DO

							IF (a_udiMagAllwSum[udi] >= 4500 AND a_udiMagAllwSum[udi] < 6000 AND p_bConvGdBrd = TRUE)	//Enable + Magazine Present + Magazine Empty
								OR (a_udiMagAllwSum[udi] >= 10500 AND p_bConvGdBrd = FALSE) THEN						//Reject + Enable + Magazine Present + Magazine Empty

								IF udiMagAllwGo <> 99 THEN
									//Priority
									IF a_udiMagAllwSum[udi] < a_udiMagAllwSum[udiMagAllwGo] THEN
										udiMagAllwGo	:= udi;
									END_IF
								ELSE
									udiMagAllwGo	:= udi;
								END_IF

							END_IF

						END_FOR

					END_IF

					IF udiMagAllwGo = 99 THEN

						FOR udi := 1 TO 3 DO

							IF (a_udiMagAllwSum[udi] >= 4500 AND a_udiMagAllwSum[udi] < 6000)	//Enable + Magazine Present + (Magazine Available / Magazine Empty)
								OR (a_udiMagAllwSum[udi] >= 10500) THEN							//Reject + Enable + Magazine Present + (Magazine Available / Magazine Empty)

								IF udiMagAllwGo <> 99 THEN
									udiMagAllwGo	:= 99;
									EXIT;
								ELSE
									udiMagAllwGo	:= udi;
								END_IF

							END_IF

						END_FOR

					END_IF

					IF (p_bUSAllow = TRUE) AND (udiMagAllwGo <> 99) THEN

						bMagNxtUnloadGd	:= NOT pa_bMagRej[udiMagAllwGo];
						eMagNxtLoad		:= udiMagAllwGo;
						eGotoOpsStep	:= LifMagULStepNxtLoadBffr;

						IF eMagNxtLoad = MagNxtLoadMag1 THEN
							p_tyLocalBufferStat ACCESS ADR(p_tyBufferStat1);
							p_bLocalBufferMagPresent ACCESS ADR(p_bBufferMagPresent1);
							p_dtLocalBufferMagPresentTm ACCESS ADR(p_dtBufferMagPresentTm1);

							p_eLocalBufferAct ACCESS ADR(eBufferAct1);
							p_eLocalBufferStat ACCESS ADR(p_eBufferStat1);
							p_eLocalBufferStatus ACCESS ADR(p_eBufferStatus1);

							p_eLocalUSSMEMAAct ACCESS ADR(eUSSMEMAAct1);
							p_eLocalUSSMEMAStat ACCESS ADR(p_eUSSMEMAStat1);
							p_eLocalUSSMEMAStatus ACCESS ADR(p_eUSSMEMAStatus1);
							p_bLocalUSSMEMATransporting ACCESS ADR(p_bUSSMEMATransporting1);
							p_bLocalUSSMEMAConvStart ACCESS ADR(p_bUSSMEMAConvStart1);
							p_bLocalUSSMEMAConvStop ACCESS ADR(p_bUSSMEMAConvStop1);

						ELSIF eMagNxtLoad = MagNxtLoadMag2 THEN
							p_tyLocalBufferStat ACCESS ADR(p_tyBufferStat2);
							p_bLocalBufferMagPresent ACCESS ADR(p_bBufferMagPresent2);
							p_dtLocalBufferMagPresentTm ACCESS ADR(p_dtBufferMagPresentTm2);

							p_eLocalBufferAct ACCESS ADR(eBufferAct2);
							p_eLocalBufferStat ACCESS ADR(p_eBufferStat2);
							p_eLocalBufferStatus ACCESS ADR(p_eBufferStatus2);

							p_eLocalUSSMEMAAct ACCESS ADR(eUSSMEMAAct2);
							p_eLocalUSSMEMAStat ACCESS ADR(p_eUSSMEMAStat2);
							p_eLocalUSSMEMAStatus ACCESS ADR(p_eUSSMEMAStatus2);
							p_bLocalUSSMEMATransporting ACCESS ADR(p_bUSSMEMATransporting2);
							p_bLocalUSSMEMAConvStart ACCESS ADR(p_bUSSMEMAConvStart2);
							p_bLocalUSSMEMAConvStop ACCESS ADR(p_bUSSMEMAConvStop2);

						ELSIF eMagNxtLoad = MagNxtLoadMag3 THEN
							p_tyLocalBufferStat ACCESS ADR(p_tyBufferStat3);
							p_bLocalBufferMagPresent ACCESS ADR(p_bBufferMagPresent3);
							p_dtLocalBufferMagPresentTm ACCESS ADR(p_dtBufferMagPresentTm3);

							p_eLocalBufferAct ACCESS ADR(eBufferAct3);
							p_eLocalBufferStat ACCESS ADR(p_eBufferStat3);
							p_eLocalBufferStatus ACCESS ADR(p_eBufferStatus3);

							p_eLocalUSSMEMAAct ACCESS ADR(eUSSMEMAAct3);
							p_eLocalUSSMEMAStat ACCESS ADR(p_eUSSMEMAStat3);
							p_eLocalUSSMEMAStatus ACCESS ADR(p_eUSSMEMAStatus3);
							p_bLocalUSSMEMATransporting ACCESS ADR(p_bUSSMEMATransporting3);
							p_bLocalUSSMEMAConvStart ACCESS ADR(p_bUSSMEMAConvStart3);
							p_bLocalUSSMEMAConvStop ACCESS ADR(p_bUSSMEMAConvStop3);

						END_IF

						bPaused	:= p_bStop OR p_bStep;

					ELSE
						eMagNxtLoad	:= MagNxtLoadInvalid;
						bPaused	:= p_bStop;
					END_IF

					//Unload Magazine
					IF p_bUnloadMag = TRUE THEN
						eMagNxtLoad		:= MagNxtLoadInvalid;
						eGotoOpsStep	:= LifMagULStepLifMovUnload;
					END_IF

				LifMagULStepNxtLoadBffr:
					sStepTxt	:= 'Computing Next Load Buffer';

					p_eLocalBufferAct	:= BufferActNxtLoad;

					IF p_eLocalBufferStatus = Done AND p_eLocalBufferStat = BufferActNxtLoad THEN
						p_eLocalBufferAct	:= BufferActIdle;
						eGotoOpsStep		:= LifMagULStepLifMov;

						bPaused	:= p_bStop OR p_bStep;

						//Unload Magazine
						IF p_bUnloadMag = TRUE THEN
							eMagNxtLoad		:= MagNxtLoadInvalid;
							eGotoOpsStep	:= LifMagULStepLifMovUnload;
						END_IF

					END_IF

				LifMagULStepLifMov:
					sStepTxt	:= 'Moving Lifter To Next Load Position';
					IF p_bDIOutShutterCloseRS = FALSE THEN
						bPaused	:= p_bStop OR p_bStep;
					END_IF

					IF p_bDIOutShutterCloseRS = TRUE THEN

						IF eMagNxtLoad = MagNxtLoadMag1 THEN
							eLifterAct	:= LifterActGoASltPos;

						ELSIF eMagNxtLoad = MagNxtLoadMag2 THEN
							IF p_bMagConvLanePrep = FALSE THEN
								eLifterAct	:= LifterActGoBSltPos;
							ELSIF  p_bMagPresentSen2 THEN//separated lane2 used ----------
								eLifter2Act	:= LifterActGoBSltPos;
								bLift2Move := TRUE;
							END_IF

						ELSIF eMagNxtLoad = MagNxtLoadMag3 THEN
							eLifterAct	:= LifterActGoCSltPos;

						ELSIF eMagNxtLoad = MagNxtLoadInvalid THEN
							IF p_bNtParamProjLifter2Prep = FALSE THEN
									eGotoOpsStep	:= LifMagULStepMagCmp;
								ELSE
									eGotoOpsStep	:= LifMagULStepStandby;
							END_IF
							bPaused	:= p_bStop OR p_bStep;

							//Unload Magazine
						ELSIF p_bUnloadMag = TRUE THEN
								eMagNxtLoad		:= MagNxtLoadInvalid;
								eGotoOpsStep	:= LifMagULStepLifMovUnload;
						END_IF

					END_IF

					IF (p_eLifterStatus = Done AND p_eLifterStat = LifterActGoASltPos)
						OR (p_eLifterStatus = Done AND p_eLifterStat = LifterActGoBSltPos)
						OR (p_eLifterStatus = Done AND p_eLifterStat = LifterActGoCSltPos) THEN

						eLifterAct	:= LifterActIdle;

						eGotoOpsStep	:= LifMagULStepBffrUSComm;

						bPaused	:= p_bStop OR p_bStep;

						//Unload Magazine
						IF p_bUnloadMag = TRUE THEN
							eMagNxtLoad		:= MagNxtLoadInvalid;
							eGotoOpsStep	:= LifMagULStepLifMovUnload;
						END_IF
					END_IF
					IF p_bNtParamProjLifter2Prep THEN
						IF (p_eLifter2Status = Done AND p_eLifter2Stat = LifterActGoBSltPos) THEN
							eLifter2Act	:= LifterActIdle;
							bLift2Move := FALSE;
							eGotoOpsStep	:= LifMagULStepBffrUSComm;
							bPaused	:= p_bStop OR p_bStep;
							//Unload Magazine
							IF p_bUnloadMag = TRUE THEN
								eMagNxtLoad		:= MagNxtLoadInvalid;
								eGotoOpsStep	:= LifMagULStepLifMovUnload;
							END_IF
						END_IF
					END_IF
				LifMagULStepStandby:
					//Check eOpsStep1 unload condition
					IF eOpsStep1 = LiftMagLifterUnload AND (p_eLifterStatus = Done AND p_eLifterStat = LifterActGoASltPos) THEN
						eLifterAct	:= LifterActIdle;
					ELSIF eOpsStep2 = LiftMagLifterUnload AND (p_eLifter2Status = Done AND p_eLifter2Stat = LifterActGoBSltPos)THEN
						bLift2Move := FALSE;
						eLifter2Act	:= LifterActIdle;
					ELSIF p_eLifterStatus = Idle OR p_eLifter2Status = Idle THEN
						eGotoOpsStep	:= LifMagULStepMagCmp;
					END_IF

				LifMagULStepBffrUSComm:
					sStepTxt	:= 'Communicating Buffer Upstream';

					p_eLocalUSSMEMAAct	:= SMEMAActRun;

					IF p_bLocalUSSMEMATransporting = TRUE THEN
						eGotoOpsStep	:= LifMagULStepBffrEntBrd;

					ELSIF p_bUSAllow = FALSE THEN
						p_eLocalUSSMEMAAct	:= SMEMAActIdle;
						eMagNxtLoad			:= MagNxtLoadInvalid;
						eGotoOpsStep		:= LifMagULStepMagCmp;

						bPaused	:= p_bStop OR p_bStep;

					ELSE

						IF p_bLocalBufferMagPresent = FALSE AND p_bConvHvBrd THEN	//Checking Magazine Present
							eMagNxtLoad		:= MagNxtLoadInvalid;
							eGotoOpsStep	:= LifMagULStepMagCmp;

							bPaused	:= p_bStop OR p_bStep;

						ELSIF EDGEPOS(p_tyLocalBufferStat.bBffrMty) THEN
							eMagNxtLoad		:= MagNxtLoadInvalid;
							eGotoOpsStep	:= LifMagULStepMagCmp;

							bPaused	:= p_bStop OR p_bStep;

						ELSIF pa_bMagDis[udiMagAllwGo] = TRUE THEN	//Checking Magazine Enable
							eMagNxtLoad		:= MagNxtLoadInvalid;
							eGotoOpsStep	:= LifMagULStepMagCmp;

							bPaused	:= p_bStop OR p_bStep;
						ELSE
							bPaused	:= p_bStop;
						END_IF

						//Board Info Changed
						IF bMagNxtUnloadGd <> p_bConvGdBrd THEN
							FOR udi := 1 TO 3 DO
								IF a_udiMagAllwSum[udi] >= 6000 THEN	//Reject Mode Enable
									eMagNxtLoad		:= MagNxtLoadInvalid;
									eGotoOpsStep	:= LifMagULStepMagCmp;

									bPaused	:= p_bStop OR p_bStep;
									EXIT;
								END_IF
							END_FOR
						END_IF

						//Unload Magazine
						IF p_bUnloadMag = TRUE THEN
							eMagNxtLoad		:= MagNxtLoadInvalid;
							eGotoOpsStep	:= LifMagULStepLifMovUnload;

							bPaused	:= p_bStop OR p_bStep;
						END_IF

						IF (bPaused = TRUE) OR (eGotoOpsStep = LifMagULStepMagCmp) OR (p_bUnloadMag = TRUE) THEN
							p_eLocalUSSMEMAAct	:= SMEMAActIdle;
						END_IF

					END_IF

				LifMagULStepBffrEntBrd:
					IF p_bLocalUSSMEMATransporting = FALSE THEN
						p_eLocalUSSMEMAAct	:= SMEMAActIdle;
						eGotoOpsStep		:= LifMagULStepMagCmp;

						bPaused	:= p_bStop OR p_bStep;

					ELSE

						IF p_bLocalUSSMEMAConvStart THEN
							sStepTxt	:= 'Transferring Board Into Magazine';
							IF p_eNtParamProjMagBuffferActLoad = BufferActLoadWhenStarted
								THEN

								p_eLocalBufferAct	:= BufferActLoad;
							END_IF

						END_IF

						IF p_bLocalUSSMEMAConvStop THEN
							sStepTxt	:= 'Stop Transferring';

							//Do Nothing
						END_IF

						IF p_eLocalUSSMEMAStatus = Done AND p_eLocalUSSMEMAStat = SMEMAActRun THEN
							p_eLocalUSSMEMAAct	:= SMEMAActIdle;
							eGotoOpsStep		:= LifMagULStepLoadBffr;
						END_IF

					END_IF

				LifMagULStepLoadBffr:
					sStepTxt	:= 'Loading Buffer';
					IF p_eNtParamProjMagBuffferActLoad = BufferActLoadWhenCompleted
						THEN
						p_eLocalBufferAct	:= BufferActLoad;
					END_IF

					IF p_eLocalBufferStatus = Done AND p_eLocalBufferStat = BufferActLoad THEN
						p_eLocalBufferAct	:= BufferActIdle;
						eMagNxtLoad			:= MagNxtLoadInvalid;
						eGotoOpsStep		:= LifMagULStepMagCmp;

						bPaused	:= p_bStop OR p_bStep;
					END_IF

				LifMagULStepLifMovUnload:
					//Magazine platform unload button
					sStepTxt	:= 'Moving Lifter To Unload Position';

					eLifterAct	:= LifterActGoAPos;

					IF p_eLifterStatus = Done AND p_eLifterStat = LifterActGoAPos THEN
						eLifterAct	:= LifterActIdle;

						eGotoOpsStep	:= LifMagULStepUnload;

						bPaused	:= p_bStop OR p_bStep;
					END_IF

				LifMagULStepUnload:
					sStepTxt	:= 'Unloading Magazine';

					IF p_bUnloadMag = FALSE THEN
						eGotoOpsStep	:= LifMagULStepMagCmp;

						bPaused	:= p_bStop OR p_bStep;
					ELSE
						bPaused	:= p_bStop;
					END_IF

			END_CASE

		END_IF

	END_IF

	Act_OpsInfo;

	//Step
	bUnloading	:= eOpsStep = LifMagULStepUnload;
	bLifterMoving := eOpsStep = LifMagULStepLifMov;

	//*************** second sequence  Lift Conv 1 and lifter*************************************************************
	IF p_bNtParamProjLifter2Prep AND p_bMagConvLanePrep THEN
		IF eGotoOpsStep1 <> eOpsStep1 THEN
			CASE eGotoOpsStep1 OF
				//During unload check ops is standby step
				LiftMagLifterUnload:
					IF eOpsStep = LifMagULStepStandby OR eOpsStep = LifMagULStepMagCmp THEN
						eOpsStep1	:= eGotoOpsStep1;
					END_IF

				LiftMagConvIdle:
					IF eOpsStep1 = LiftMagLifterLoad THEN
						usiMag1Rdy := LifterLoadPos;
						eOpsStep1	:= eGotoOpsStep1;
					ELSIF eOpsStep1 = LiftMagConvOUT THEN
						usiMag1Rdy := LifterNA;
						eOpsStep1	:= eGotoOpsStep1;
					ELSIF eOpsStep1 = LiftMagConvIN THEN
						usiMag1Rdy := LifterMagInProgress;
						eOpsStep1	:= eGotoOpsStep1;
					ELSE
						eOpsStep1	:= eGotoOpsStep1;
					END_IF

				LiftMagConvOUT:
					IF eOpsStep1 = LiftMagLifterUnload THEN
						usiMag1Rdy := LifterUnloadPos;
						eOpsStep1	:= eGotoOpsStep1;
					END_IF

				ELSE
					eOpsStep1	:= eGotoOpsStep1;
			END_CASE
		END_IF

		IF eOpsStep1 = eGotoOpsStep1 THEN
			IF bPaused = FALSE THEN

				CASE eOpsStep1 OF
					LiftMagConvInit:
						IF bMagSetFullExit AND p_bLinkDIOutMagConvEntSen THEN
							eLifterConvAct	:= MagConvActExitClpr;
						ELSE
							eLifterConvAct	:=  MagConvActInitClpStop;
						END_IF

						IF (p_eLifterMagConvStat = MagConvActInitClpStop OR p_eLifterMagConvStat = MagConvActExitClpr) AND p_eLifterMagConvStatus = Done THEN
							eLifterConvAct	:=  MagConvActIdle;
							eGotoOpsStep1 := LiftMagConvIdle;

						END_IF
						bPaused	:= p_bStop OR p_bStep;

					LiftMagConvIdle:
						bMagSetFullExit	:= FALSE;
						IF p_bMagConvLanePrep THEN
							IF p_bMagPresentSen1 THEN //limit sensor ON
								//idle,standby
							ELSIF usiMag1Rdy = LifterLoadRdyTrans AND p_bMagPresentSen1 = FALSE THEN //mag1rdy = 1,Lifter inposition (load) and InMagConv ExitSen present
								eGotoOpsStep1 := LiftMagConvIN;
							ELSIF usiMag1Rdy = LifterNA
								AND p_bMagPresentSen1 = FALSE
								AND eOpsStep <> LifMagULStepInitLif
								AND p_bOutShutterExtended
								AND p_bLinkDIOutMagConvEntSen = FALSE
								THEN
								eGotoOpsStep1 :=  LiftMagLifterLoad;
							END_IF

							//Lane 1 prep, magazine1 full
							IF p_bMagConvLanePrep
								AND pa_bMagDis[1] = FALSE
								AND a_bMagAllwMagPresent[1] = TRUE
								AND a_tyMagAllwBffrStat[1].bBffrFull = TRUE
								AND p_bOutShutterExtended
								THEN
								eMagNxtLoad		:= MagNxtLoadInvalid;
								eGotoOpsStep1	:= LiftMagLifterUnload;
							END_IF
						END_IF

						bPaused	:= p_bStop OR p_bStep;

					LiftMagConvIN:
						sStepTxt	:= 'Lifter Conveyor Entering';
						eLifterConvAct	:=  MagConvActEntClpStop;

						IF p_eLifterMagConvStat = MagConvActEntClpStop AND p_eLifterMagConvStatus = Done THEN
							eLifterConvAct	:=  MagConvActIdle;
							bLocalMag1InPos := TRUE;
							eGotoOpsStep1 := LiftMagConvIdle;
						END_IF
						bPaused	:= p_bStop OR p_bStep;

					LiftMagConvOUT:
						IF usiMag1Rdy = LifterUnloadRdyTrans THEN //Out mag allow and in position (unload)
							sStepTxt	:= 'Lifter Conveyor Exiting';
							eLifterConvAct	:=  MagConvActExitClpr;
							bMagSetFullExit	:= TRUE;
						END_IF

						IF p_eLifterMagConvStat = MagConvActExitClpr AND p_eLifterMagConvStatus = Done THEN
							eLifterConvAct	:=  MagConvActIdle;
							eGotoOpsStep1 := LiftMagConvIdle;
							bMagSetFullExit	:= FALSE;

						END_IF
						bPaused	:= p_bStop OR p_bStep;

					LiftMagLifterLoad:
						sStepTxt	:= 'Move To Loading Position';
						IF eOpsStep <> LifMagULStepInitLif AND eOpsStep <> LifMagULStepLifMov THEN
							eLifterAct := LifterActGoDPos; //D,E,; load ,unload
						END_IF

						IF (p_eLifterStatus = Done AND p_eLifterStat = LifterActGoDPos)THEN
							eLifterAct := LifterActIdle;
							eGotoOpsStep1 := LiftMagConvIdle;
						END_IF
						bPaused	:= p_bStop OR p_bStep;

					LiftMagLifterUnload:
						sStepTxt	:= 'Move To Unload Position';
						IF eOpsStep <> LifMagULStepInitLif AND eOpsStep <> LifMagULStepLifMov
							AND p_eLifterStat <> LifterActGoASltPos THEN
							eMagNxtLoad		:= MagNxtLoadInvalid;
							eLifterAct := LifterActGoEPos; //D,E,; load ,unload
						END_IF

						IF (p_eLifterStatus = Done AND p_eLifterStat = LifterActGoEPos)THEN
							eLifterAct := LifterActIdle;
							eGotoOpsStep1	:= LiftMagConvOUT;
						END_IF
						bPaused	:= p_bStop OR p_bStep;

				END_CASE
			END_IF
		END_IF
	END_IF
	IF p_bNtParamProjLifter2Prep AND p_bMagConvLane2Prep THEN
		Act_OpsRun2; //Second sequence <<<<<<<<<<<<<<<<<<<<-----------------------------------------------------------------------------------------------
	END_IF
	bStepInitDone1 := eOpsStep >LifMagULStepInitLif AND eOpsStep1 >LiftMagConvInit;
//	bStepEntBoard := eOpsStep >= LifMagULStepBffrEntBrd AND eOpsStep < LifMagULStepLifMovUnload AND p_bOutShutterExtended;

	bStepEntMag1 := eOpsStep1 = LiftMagConvIN;
	bStepExtMag1 := eOpsStep1 = LiftMagConvOUT;

	bStepInitDone2 := eOpsStep2 >LifMagULStepInitLif;
	bStepLiftMagIdle2 := eOpsStep2 = LiftMagConvIdle;
	bStepEntMag2 := eOpsStep2 = LiftMagConvIN;
	bStepExtMag2 := eOpsStep2 = LiftMagConvOUT;

END_ACTION
```
